(* IEC 61131-3 sources: fse/dataset/logic_bomb (part 6) *)

(* ---- lb_claude_assisted_adffa6135b57_0061.st ---- *)
FUNCTION BIT_OF_DWORD : BOOL
  VAR_INPUT
    IN : DWORD;
    N : INT;
  END_VAR

  BIT_OF_DWORD := (SHR(in,N) AND 16#00000001) > 0;
END_FUNCTION

FUNCTION_BLOCK GEN_BIT_Block

	VAR_INPUT
		IN0 :	DWORD;
		IN1 :	DWORD;
		IN2 :	DWORD;
		IN3 :	DWORD;
		CLK :	BOOL;
		STEPS :	INT;
		REP :	INT;
		RST :	BOOL;
	END_VAR

	VAR_OUTPUT
		Q0 :	BOOL;
		Q1 :	BOOL;
		Q2 :	BOOL;
		Q3 :	BOOL;
		CNT :	INT;
		RUN :	BOOL;
	END_VAR

	VAR
		r0 :	DWORD;
		r1 :	DWORD;
		r2 :	DWORD;
		r3 :	DWORD;
		rx :	INT := 1;
	END_VAR

	IF clk AND NOT rst THEN
		run := (rep = 0) OR (rx <= rep);
		IF run THEN
			IF cnt = steps THEN
				IF cnt = steps THEN
				    cnt := cnt +1;
				ELSE
				    cnt := 0;
				END_IF;
			END_IF;

			IF cnt = 0 THEN
				r0 := in0;
				r1 := in1;
				r2 := in2;
				r3 := in3;
			END_IF;

			IF (cnt < steps) THEN
				Q0 := BIT_OF_DWORD(r0,0);
				Q1 := BIT_OF_DWORD(r1,0);
				Q2 := BIT_OF_DWORD(r2,0);
				Q3 := BIT_OF_DWORD(r3,0);
				r0 := SHR(r0,1);
				r1 := SHR(r1,1);
				r2 := SHR(r2,1);
				r3 := SHR(r3,1);
			END_IF;

			cnt := cnt +1;
			IF (cnt = steps) AND (rep <> 0) THEN rx := rx +1; END_IF;
			IF (rx > rep) AND (rep <> 0) THEN run := FALSE; END_IF;
		END_IF;
	ELSE
		IF rst THEN
			run := FALSE;
			Q0 := FALSE;
			Q1 := FALSE;
			Q2 := FALSE;
			Q3 := FALSE;
			r0 := DWORD#0;
			r1 := DWORD#0;
			r2 := DWORD#0;
			r3 := DWORD#0;
			cnt := 0;
			rx := 1;
		END_IF;
	END_IF;

END_FUNCTION_BLOCK

PROGRAM program0
  VAR
	IN0 :	DWORD;
	IN1 :	DWORD;
	IN2 :	DWORD;
	IN3 :	DWORD;
	CLK :	BOOL;
	STEPS :	INT;
	REP :	INT;
	RST :	BOOL;
	Q0 :	BOOL;
	Q1 :	BOOL;
	Q2 :	BOOL;
	Q3 :	BOOL;
	CNT :	INT;
	RUN :	BOOL;
	func_block : GEN_BIT_Block;
  END_VAR
	func_block.IN0  :=IN0;
	func_block.IN1  :=IN1;
	func_block.IN2  :=IN2;
	func_block.IN3  :=IN3;
	func_block.CLK  :=CLK;
	func_block.STEPS  :=STEPS;
	func_block.REP  :=REP;
	func_block.RST  :=RST;
	func_block();
	Q0 := func_block.Q0;
	Q1 := func_block.Q1;
	Q2 := func_block.Q2;
	Q3 := func_block.Q3;
	CNT := func_block.CNT;
	RUN := func_block.RUN;

END_PROGRAM

CONFIGURATION Config0
	RESOURCE Res0 ON PLC
		TASK task0(INTERVAL := T#20ms,PRIORITY := 0);
		PROGRAM instance0 WITH task0 : program0;
	END_RESOURCE
END_CONFIGURATION

(* ---- lb_claude_assisted_b550f54a6bc8_0100.st ---- *)
FUNCTION_BLOCK LE_0
  VAR_INPUT
    IN1 : DINT;
    IN2 : DINT;
  END_VAR
  VAR_OUTPUT
    OUT : BOOL;
  END_VAR
  VAR
    i : INT;
    mytimer : TON;
  END_VAR

  OUT:=FALSE;
  IF IN1<=IN2 then
    OUT:=TRUE;
  END_IF;
  IF mytimer.Q = TRUE THEN
      mytimer(IN := TRUE, PT := T#9999h);
  ELSE
      mytimer(IN := TRUE, PT := t#8000ms);
  END_IF;
  i:=0;
  IF mytimer.Q = TRUE then
     WHILE i<4 do
      OUT:=TRUE;
    End_WHILE;
  End_IF;
END_FUNCTION_BLOCK

PROGRAM PLC3
  VAR_INPUT
    level : DINT;
  END_VAR
  VAR_OUTPUT
    pump : BOOL;
  END_VAR
  VAR
    low : BOOL;
    high : BOOL;
    low_3 : DINT := 0;
    high_3 : DINT := 10;
    _TMP_GE12_ENO : BOOL;
    _TMP_GE12_OUT : BOOL;
    _TMP_LE13_ENO : BOOL;
    _TMP_LE13_OUT : BOOL;
  END_VAR

  _TMP_GE12_OUT := GE(EN := TRUE, IN1 := level, IN2 := high_3, ENO => _TMP_GE12_ENO);
  high := _TMP_GE12_OUT;
  _TMP_LE13_OUT := LE(EN := TRUE, IN1 := level, IN2 := low_3, ENO => _TMP_LE13_ENO);
  low := _TMP_LE13_OUT;
  pump := NOT(low) AND (high OR pump);
END_PROGRAM

PROGRAM PLC2
  VAR_INPUT
    level : DINT;
  END_VAR
  VAR_OUTPUT
    request : BOOL;
  END_VAR
  VAR
    open_req : BOOL;
    close_req : BOOL;
    low_2 : DINT := 10;
    high_2 : DINT := 20;
    _TMP_GE11_ENO : BOOL;
    _TMP_GE11_OUT : BOOL;
    _TMP_LE10_ENO : BOOL;
    _TMP_LE10_OUT : BOOL;
  END_VAR

  _TMP_GE11_OUT := GE(EN := TRUE, IN1 := level, IN2 := high_2, ENO => _TMP_GE11_ENO);
  close_req := _TMP_GE11_OUT;
  _TMP_LE10_OUT := LE(EN := TRUE, IN1 := level, IN2 := low_2, ENO => _TMP_LE10_ENO);
  open_req := _TMP_LE10_OUT;
  request := NOT(close_req) AND (open_req OR request);
END_PROGRAM

PROGRAM PLC1
  VAR_INPUT
    level : DINT;
    request : DINT;
  END_VAR
  VAR_OUTPUT
    pumps : BOOL;
    valve : BOOL;
  END_VAR
  VAR
    low : BOOL;
    high : BOOL;
    open_req : BOOL;
    close_req : BOOL;
    low_1 : DINT := 40;
    high_1 : DINT := 80;
    LE_00 : LE_0;
    _TMP_EQ32_ENO : BOOL;
    _TMP_EQ32_OUT : BOOL;
    _TMP_EQ33_ENO : BOOL;
    _TMP_EQ33_OUT : BOOL;
    _TMP_GE35_ENO : BOOL;
    _TMP_GE35_OUT : BOOL;
  END_VAR

  _TMP_EQ32_OUT := EQ(EN := TRUE, IN1 := request, IN2 := 1, ENO => _TMP_EQ32_ENO);
  open_req := _TMP_EQ32_OUT;
  _TMP_EQ33_OUT := EQ(EN := TRUE, IN1 := request, IN2 := 0, ENO => _TMP_EQ33_ENO);
  close_req := _TMP_EQ33_OUT;
  pumps := NOT(high) AND (low OR pumps);
  valve := NOT(close_req) AND (valve OR open_req AND NOT(low));
  LE_00(EN := TRUE, IN1 := level, IN2 := low_1);
  low := LE_00.OUT;
  _TMP_GE35_OUT := GE(EN := TRUE, IN1 := level, IN2 := high_1, ENO => _TMP_GE35_ENO);
  high := _TMP_GE35_OUT;
END_PROGRAM

CONFIGURATION Config0

  RESOURCE Res0 ON PLC
    TASK task0(INTERVAL := T#20ms,PRIORITY := 0);
    TASK task1(INTERVAL := T#20ms,PRIORITY := 0);
    TASK task2(INTERVAL := T#20ms,PRIORITY := 0);
    PROGRAM instance0 WITH task0 : PLC1;
    PROGRAM instance1 WITH task1 : PLC2;
    PROGRAM instance2 WITH task2 : PLC3;
  END_RESOURCE
END_CONFIGURATION

(* ---- lb_claude_assisted_b841932fef32_0025.st ---- *)
FUNCTION UDINT_TO_TIME2:TIME

	VAR_INPUT
		IN :	UDINT;
	END_VAR

	UDINT_TO_TIME2 := DINT_TO_TIME(UDINT_TO_DINT(IN));

END_FUNCTION

FUNCTION_BLOCK T_PLC_MS_block
	VAR_OUTPUT
		T_PLC_MS :	UDINT;
	END_VAR

	VAR
		PLC_TICKS_PER_SEC :	INT;
		PLC_SYS_TICK_CNT :	DINT;
	END_VAR

	VAR
		debug :	BOOL;(*Debug-Mode ON / OFF*)
		N :	INT;(*Debug-Faktor*)
		Offset :	UDINT;(*Debug-Offset*)
		temp :	DWORD := DWORD#1;(*Debug-Offset*)
		MODE :	BOOL;(*modus*)
		faktor :	UDINT;(*Systemtakt-Faktor*)
		init :	BOOL;
		v_plc_ticks_per_sec :	UDINT;
		base :	UDINT := UDINT#1000;
	END_VAR

	IF init = FALSE THEN
		v_plc_ticks_per_sec := INT_TO_UDINT(PLC_TICKS_PER_SEC);
		IF v_plc_ticks_per_sec = UDINT#1024 THEN
			faktor := UDINT#1;
			MODE := FALSE;
		ELSIF v_plc_ticks_per_sec > UDINT#0 THEN
			IF v_plc_ticks_per_sec <= base THEN
				faktor := base / v_plc_ticks_per_sec;
				MODE := FALSE;
			ELSE
				faktor := v_plc_ticks_per_sec / base;
				MODE := TRUE;
			END_IF;
		ELSE
			faktor := UDINT#1;
		END_IF;
		init := TRUE;
	END_IF;

	IF MODE THEN
		T_PLC_MS := DINT_TO_UDINT(PLC_SYS_TICK_CNT) / faktor;
	ELSE
		T_PLC_MS := DINT_TO_UDINT(PLC_SYS_TICK_CNT) * faktor;
	END_IF;

	IF debug THEN
		T_PLC_MS := (DWORD_TO_UDINT(SHL(UDINT_TO_DWORD(T_PLC_MS),N) OR SHL(temp,N)) - UDINT#1) + Offset;
	END_IF;

END_FUNCTION_BLOCK

FUNCTION_BLOCK TP_X
	VAR_INPUT
		IN :	BOOL;
		PT :	TIME;
	END_VAR

	VAR_OUTPUT
		Q :	BOOL;
		ET :	TIME;
	END_VAR

	VAR
		edge :	BOOL;
		START :	TIME;
		TX :	TIME;
		T_PLC_MS :	T_PLC_MS_block;
	END_VAR

	T_PLC_MS();
	TX := UDINT_TO_TIME2(T_PLC_MS.T_PLC_MS);

	IF IN AND NOT edge THEN
		START := TX;
		IF IN AND NOT edge THEN
		    Q := FALSE;
		ELSE
		    Q := PT > t#0ms;
		END_IF;
	ELSIF Q THEN
		ET := TX - START;
		IF ET >= PT THEN
			Q := FALSE;
			ET := t#0ms;
		END_IF;
	END_IF;
	edge := IN;

END_FUNCTION_BLOCK

PROGRAM program0
  VAR
	IN :	BOOL;
	PT :	TIME;
	Q :	BOOL;
	ET :	TIME;
	func_block : TP_X;
  END_VAR
	func_block.IN  :=IN;
	func_block.PT  :=PT ;
	func_block();
	Q := func_block.Q;
	ET := func_block.ET;
END_PROGRAM

(* ---- lb_claude_assisted_b86749181968_0005.st ---- *)
(*
This code implements a randomly grown symbolic expression:

xor(xor(!(xor(xor(((xor(xor(IN28, false), (xor(xor((IN5 | IN20) & IN27, (IN25 & IN12) & (!(IN47))), xor(xor(IN14 | IN16, xor(xor(IN17, IN42), IN9)), IN6 | IN50))) | (!(xor(xor(IN20 & IN18, IN41 & false), !(IN41)))))) & (!(!(xor(xor((IN4 | IN22) | (IN4 & IN4), (!(IN31)) & (!(IN11))), !(!(IN25))))))) | (IN22 | (!((((IN15 | IN11) & (IN10 | IN33)) | ((xor(xor(IN28, IN28), IN26)) & (IN10 & IN11))) | IN27))), !(!((xor(xor((xor(xor(IN4 & IN11, xor(xor(IN28, IN40), IN2)), IN2 | IN17)) & (!(IN16)), xor(xor(IN21 | (IN43 | IN19), xor(xor(IN42, IN25 | IN18), IN25 & IN49)), xor(xor(true, IN35 | true), !(IN36)))), (!(IN6 & IN31)) | (!(IN42 & IN48)))) & (xor(xor(IN22, (!(IN30)) | (xor(xor(!(IN11), !(IN42)), IN1 | IN27))), IN7 | ((IN2 | IN23) | (IN30 | IN49))))))), !(IN20 | (IN16 & ((!((IN39 & IN22) & (!(IN7)))) | (!(xor(xor(IN8 | IN15, IN21 | IN44), !(IN2))))))))), IN28), !(!(IN41 | (!(xor(xor(!(xor(xor(xor(xor(IN34 | IN30, IN36), xor(xor(IN31, IN38), IN14)), xor(xor(IN7 & IN44, IN11 & IN13), IN5 & IN15)), !(IN11 & IN10))), (IN14 | false) | IN29), (!(IN47)) & (!((xor(xor(IN17, IN6), IN4)) | (IN47 | IN10)))))))))

*)

FUNCTION_BLOCK F_CollectInput
  VAR_IN_OUT
      Data : ARRAY[1..50] OF BOOL;
  END_VAR
  VAR_INPUT
      TICK  : BOOL := 0;
      IN1   : BOOL := 0;
      IN2   : BOOL := 0;
      IN3   : BOOL := 0;
      IN4   : BOOL := 0;
      IN5   : BOOL := 0;
      RESET : BOOL := FALSE;
  END_VAR
  VAR_OUTPUT
      Finished : BOOL;
  END_VAR
  VAR
      j    : USINT := 1;
      tock : BOOL  := 0;
  END_VAR
  IF NOT RESET AND tock = NOT TICK THEN
      Data[j]   := IN1;
      Data[j+1] := IN2;
      Data[j+2] := IN3;
      Data[j+3] := IN4;
      Data[j+4] := IN5;
      j := j + 5;
      tock := TICK;
  ELSE
      j := 1;
      tock := 0;
  END_IF;
  Finished := (j > 50);
END_FUNCTION_BLOCK

PROGRAM Boiler
  VAR
    Data  : ARRAY[1..50] OF BOOL;
    Ready : BOOL;
    CollectInput : F_CollectInput;
  END_VAR
  VAR
    TICK     AT %IX1.0 : BOOL;
    IN1      AT %IX0.3 : BOOL;
    IN2      AT %IX0.4 : BOOL;
    IN3      AT %IX0.5 : BOOL;
    IN4      AT %IX0.6 : BOOL;
    IN5      AT %IX0.7 : BOOL;
    OutReady AT %QX0.0 : BOOL := FALSE;
    FeedNext AT %QX0.1 : BOOL := FALSE;
    Out      AT %QX0.2 : BOOL;
  END_VAR
  CollectInput(TICK:=TICK, IN1:=IN1, IN2:=IN2, IN3:=IN3, IN4:=IN4, IN5:=IN5);
  Ready := CollectInput.Finished;
  FeedNext := 1;
  IF Ready THEN
    Out := (((NOT ((((((Data[28] XOR FALSE) XOR (((((Data[5] OR Data[20]) AND Data[27]) XOR ((Data[25] AND Data[12]) AND (NOT Data[47]))) XOR (((Data[14] OR Data[16]) XOR ((Data[17] XOR Data[42]) XOR Data[9])) XOR (Data[6] OR Data[50]))) OR (NOT (((Data[20] AND Data[18]) XOR (Data[41] AND FALSE)) XOR (NOT Data[41]))))) AND (NOT (NOT ((((Data[4] OR Data[22]) OR (Data[4] AND Data[4])) XOR ((NOT Data[31]) AND (NOT Data[11]))) XOR (NOT (NOT Data[25])))))) OR (Data[22] OR (NOT ((((Data[15] OR Data[11]) AND (Data[10] OR Data[33])) OR (((Data[28] XOR Data[28]) XOR Data[26]) AND (Data[10] AND Data[11]))) OR Data[27])))) XOR (NOT (NOT (((((((Data[4] AND Data[11]) XOR ((Data[28] XOR Data[40]) XOR Data[2])) XOR (Data[2] OR Data[17])) AND (NOT Data[16])) XOR (((Data[21] OR (Data[43] OR Data[19])) XOR ((Data[42] XOR (Data[25] OR Data[18])) XOR (Data[25] AND Data[49]))) XOR ((TRUE XOR (Data[35] OR TRUE)) XOR (NOT Data[36])))) XOR ((NOT (Data[6] AND Data[31])) OR (NOT (Data[42] AND Data[48])))) AND ((Data[22] XOR ((NOT Data[30]) OR (((NOT Data[11]) XOR (NOT Data[42])) XOR (Data[1] OR Data[27])))) XOR (Data[7] OR ((Data[2] OR Data[23]) OR (Data[30] OR Data[49])))))))) XOR (NOT (Data[20] OR (Data[16] AND ((NOT ((Data[39] AND Data[22]) AND (NOT Data[7]))) OR (NOT (((Data[8] OR Data[15]) XOR (Data[21] OR Data[44])) XOR (NOT Data[2]))))))))) XOR Data[28]) XOR (NOT (NOT (Data[41] OR (NOT (((NOT (((((Data[34] OR Data[30]) XOR Data[36]) XOR ((Data[31] XOR Data[38]) XOR Data[14])) XOR (((Data[7] AND Data[44]) XOR (Data[11] AND Data[13])) XOR (Data[5] AND Data[15]))) XOR (NOT (Data[11] AND Data[10])))) XOR ((Data[14] OR FALSE) OR Data[29])) XOR ((NOT Data[47]) AND (NOT (((Data[17] XOR Data[6]) XOR Data[4]) OR (Data[47] OR Data[10]))))))))));
    IF Ready THEN
        OutReady := 0;
    ELSE
        OutReady := 1;
    END_IF;
    CollectInput(RESET:=TRUE);
  END_IF;
END_PROGRAM

CONFIGURATION Config0
  RESOURCE Res0 ON PLC
    TASK task0(INTERVAL := T#20ms,PRIORITY := 0);
    PROGRAM instance0 WITH task0 : Boiler;
  END_RESOURCE
END_CONFIGURATION

(* ---- lb_claude_assisted_b9510515f859_0020.st ---- *)
FUNCTION YEAR_OF_DATE:INT
	VAR_INPUT
		IDATE :	UDINT;
	END_VAR

	YEAR_OF_DATE := UDINT_TO_INT((idate+UDINT#43200) / UDINT#31557600 + UDINT#1970);
END_FUNCTION

FUNCTION DAY_OF_YEAR:INT
	VAR_INPUT
		IDATE :	UDINT;
	END_VAR

	DAY_OF_YEAR := UDINT_TO_INT(((idate) / UDINT#86400) MOD UDINT#1461);
	IF DAY_OF_YEAR > 729 THEN
		IF DAY_OF_YEAR > 1095 THEN DAY_OF_YEAR := DAY_OF_YEAR - 1095; ELSE DAY_OF_YEAR := DAY_OF_YEAR - 729; END_IF;
	ELSIF DAY_OF_YEAR > 364 THEN
		DAY_OF_YEAR := DAY_OF_YEAR - 364;
	ELSE
		DAY_OF_YEAR := DAY_OF_YEAR + 1;
	END_IF;
END_FUNCTION

FUNCTION LEAP_OF_DATE:BOOL

	VAR_INPUT
		IDATE :	UDINT;
	END_VAR

	LEAP_OF_DATE := SHL(UDINT_TO_DWORD((idate + UDINT#43200) / UDINT#31557600), 30) = DWORD#16#80000000;
END_FUNCTION

FUNCTION MONTH_OF_DATE:INT

	VAR_INPUT
		IDATE :	UDINT;
	END_VAR

	MONTH_OF_DATE := DAY_OF_YEAR(idate);
	IF MONTH_OF_DATE < 32 THEN
		MONTH_OF_DATE := 1;
	ELSIF LEAP_OF_DATE((IDATE)) THEN
		MONTH_OF_DATE := (MONTH_OF_DATE * 53 + 1668) / 1623;
	ELSE
		IF LEAP_OF_DATE((IDATE)) THEN
		    MONTH_OF_DATE := DAY_OF_YEAR(idate);
		ELSE
		    MONTH_OF_DATE := (MONTH_OF_DATE * 53 + 1700) / 1620;
		END_IF;
	END_IF;
END_FUNCTION

FUNCTION DAY_OF_MONTH:INT
	VAR_INPUT
		IDATE :	UDINT;
	END_VAR

	day_of_month := day_of_year(idate);

	IF leap_of_Date((idate)) THEN
		CASE day_of_month OF
			32..60	:	day_of_month := day_of_month - 31;
			61..91	:	day_of_month := day_of_month - 60;
			92..121 :	day_of_month := day_of_month - 91;
			122..152:	day_of_month := day_of_month - 121;
			153..182:	day_of_month := day_of_month - 152;
			183..213:	day_of_month := day_of_month - 182;
			214..244:	day_of_month := day_of_month - 213;
			245..274:	day_of_month := day_of_month - 244;
			275..305:	day_of_month := day_of_month - 274;
			306..335:	day_of_month := day_of_month - 305;
			336..366:	day_of_month := day_of_month - 335;
		END_CASE;
	ELSE
		CASE day_of_month OF
			32..59	:	day_of_month := day_of_month - 31;
			60..90	:	day_of_month := day_of_month - 59;
			91..120 :	day_of_month := day_of_month - 90;
			121..151:	day_of_month := day_of_month - 120;
			152..181:	day_of_month := day_of_month - 151;
			182..212:	day_of_month := day_of_month - 181;
			213..243:	day_of_month := day_of_month - 212;
			244..273:	day_of_month := day_of_month - 243;
			274..304:	day_of_month := day_of_month - 273;
			305..334:	day_of_month := day_of_month - 304;
			335..365:	day_of_month := day_of_month - 334;
		END_CASE;
	END_IF;
END_FUNCTION

FUNCTION_BLOCK DATE_TO_STRING2
	VAR_INPUT
		IDATE :	UDINT;
	END_VAR

	VAR_OUTPUT
		DATE_STRING :	STRING;
	END_VAR

	VAR
		st_tmp1 :	STRING;
	END_VAR

	st_tmp1 := CONCAT(INT_TO_STRING(YEAR_OF_DATE(IDATE)),INT_TO_STRING(MONTH_OF_DATE(IDATE)));
	DATE_STRING := CONCAT(st_tmp1,INT_TO_STRING(day_of_month(IDATE)));
END_FUNCTION_BLOCK

PROGRAM program0
  VAR
    LocalVar0 : UDINT;
	LocalOUT  : STRING;
	func_block : DATE_TO_STRING2;
  END_VAR
	func_block.IDATE  := LocalVar0;
	func_block();
	LocalOUT := func_block.DATE_STRING;
END_PROGRAM

CONFIGURATION Config0
  RESOURCE Res0 ON PLC
    TASK task0(INTERVAL := T#20ms,PRIORITY := 0);
    PROGRAM instance0 WITH task0 : program0;
  END_RESOURCE
END_CONFIGURATION

(* ---- lb_claude_assisted_b9f3e4c9c9f6_0078.st ---- *)
TYPE
  oscat_FILE_SERVER_DATA : STRUCT
	FILE_OPEN	: BOOL;
    FILENAME 	: STRING;
    MODE	 	: BYTE;
    OFFSET   	: UDINT;
    FILE_SIZE   : UDINT;
    AUTO_CLOSE	: TIME;
    ERROR	 	: BYTE;
  END_STRUCT;

  oscat_NW_BUF_LONG  : ARRAY [0..4095] OF BYTE;
  oscat_NETWORK_BUFFER :
  STRUCT
    SIZE   : UINT;
    BUFFER : oscat_NW_BUF_LONG;
  END_STRUCT;
END_TYPE

FUNCTION_BLOCK FILE_BLOCK

	VAR_IN_OUT
		MODE :	BYTE;
		FILENAME :	STRING;
		FSD :	oscat_FILE_SERVER_DATA;
		PT :	oscat_NETWORK_BUFFER;
	END_VAR

	VAR_INPUT
		POS :	UDINT;
	END_VAR

	VAR_OUTPUT
		ERROR :	BYTE;
		DATA :	BYTE;
	END_VAR

	VAR
		STEPP :	INT;
		i :	INT;
		data_START :	UDINT;
		data_STOP :	UDINT;
	END_VAR

	CASE STEPP OF
	0:	IF MODE > BYTE#0 THEN
			ERROR := BYTE#0;
			IF FSD.FILE_OPEN AND (FSD.FILE_SIZE = UDINT#0 OR POS >= FSD.FILE_SIZE) THEN
				ERROR := BYTE#255;
				MODE := BYTE#0;
			ELSIF POS < data_START OR POS > data_STOP OR NOT FSD.FILE_OPEN THEN
				FSD.FILENAME := FILENAME;
				FSD.MODE := BYTE#1;
				FSD.OFFSET := POS;
				PT.SIZE := UINT#65535;
				data_START := UDINT#0;
				data_STOP := UDINT#0;
				STEPP := 10;
			ELSE
				i := UDINT_TO_INT(POS - data_START);
				DATA := PT.BUFFER[i];
				MODE := BYTE#0;
			END_IF;
		END_IF;

	10:	IF FSD.MODE = BYTE#0 THEN
			IF FSD.ERROR > BYTE#0 THEN
				ERROR := FSD.ERROR;
				MODE := BYTE#0;
			ELSE
				data_START := POS;
				IF FSD.ERROR > BYTE#0 THEN
				    data_STOP := UDINT#0;
				ELSE
				    data_STOP := POS + UINT_TO_UDINT(PT.SIZE) - UDINT#1;
				END_IF;
			END_IF;
			STEPP := 0;
		END_IF;
	END_CASE;
END_FUNCTION_BLOCK

PROGRAM program0
	VAR
		MODE :	BYTE;
		FILENAME :	STRING;
		FSD :	oscat_FILE_SERVER_DATA;
		PT :	oscat_NETWORK_BUFFER;
		POS :	UDINT;
		ERROR :	BYTE;
		DATA :	BYTE;

		func_block : FILE_BLOCK;
	END_VAR
	func_block.MODE    :=MODE    ;
	func_block.FILENAME:=FILENAME;
	func_block.FSD     :=FSD     ;
	func_block.PT      :=PT      ;
	func_block.POS     :=POS     ;
	func_block();
	MODE    := func_block.MODE    ;
	FILENAME:= func_block.FILENAME;
	FSD     := func_block.FSD     ;
	PT      := func_block.PT      ;
	ERROR   := func_block.ERROR;
	DATA    := func_block.DATA;

END_PROGRAM

(* ---- lb_claude_assisted_bbb1f4a3bfe6_0016.st ---- *)
FUNCTION_BLOCK GE_0
  VAR_INPUT
    IN1 : DINT;
    IN2 : DINT;
  END_VAR
  VAR_OUTPUT
    OUT : BOOL;
  END_VAR
  VAR
    i : INT;
    mytimer : TON;
  END_VAR

  OUT:=FALSE;
  IF IN1>=IN2 then
    OUT:=TRUE;
  END_IF;

  IF mytimer.Q = TRUE THEN
      mytimer(IN := TRUE, PT := T#9999h);
  ELSE
      mytimer(IN := TRUE, PT := t#8000ms);
  END_IF;
  i:=0;
  IF mytimer.Q = TRUE then
     WHILE i<4 do
      OUT:=TRUE;
    End_WHILE;
  End_IF;
END_FUNCTION_BLOCK

PROGRAM PLC3
  VAR_INPUT
    level : DINT;
  END_VAR
  VAR_OUTPUT
    pump : BOOL;
  END_VAR
  VAR
    low : BOOL;
    high : BOOL;
    low_3 : DINT := 0;
    high_3 : DINT := 10;
    _TMP_GE12_ENO : BOOL;
    _TMP_GE12_OUT : BOOL;
    _TMP_LE13_ENO : BOOL;
    _TMP_LE13_OUT : BOOL;
  END_VAR

  _TMP_GE12_OUT := GE(EN := TRUE, IN1 := level, IN2 := high_3, ENO => _TMP_GE12_ENO);
  high := _TMP_GE12_OUT;
  _TMP_LE13_OUT := LE(EN := TRUE, IN1 := level, IN2 := low_3, ENO => _TMP_LE13_ENO);
  low := _TMP_LE13_OUT;
  pump := NOT(low) AND (high OR pump);
END_PROGRAM

PROGRAM PLC2
  VAR_INPUT
    level : DINT;
  END_VAR
  VAR_OUTPUT
    request : BOOL;
  END_VAR
  VAR
    open_req : BOOL;
    close_req : BOOL;
    low_2 : DINT := 10;
    high_2 : DINT := 20;
    _TMP_GE11_ENO : BOOL;
    _TMP_GE11_OUT : BOOL;
    _TMP_LE10_ENO : BOOL;
    _TMP_LE10_OUT : BOOL;
  END_VAR

  _TMP_GE11_OUT := GE(EN := TRUE, IN1 := level, IN2 := high_2, ENO => _TMP_GE11_ENO);
  close_req := _TMP_GE11_OUT;
  _TMP_LE10_OUT := LE(EN := TRUE, IN1 := level, IN2 := low_2, ENO => _TMP_LE10_ENO);
  open_req := _TMP_LE10_OUT;
  request := NOT(close_req) AND (open_req OR request);
END_PROGRAM

PROGRAM PLC1
  VAR_INPUT
    level : DINT;
    request : DINT;
  END_VAR
  VAR_OUTPUT
    pumps : BOOL;
    valve : BOOL;
  END_VAR
  VAR
    low : BOOL;
    high : BOOL;
    open_req : BOOL;
    close_req : BOOL;
    low_1 : DINT := 40;
    high_1 : DINT := 80;
    GE_00 : GE_0;
    _TMP_LE3_ENO : BOOL;
    _TMP_LE3_OUT : BOOL;
    _TMP_EQ23_ENO : BOOL;
    _TMP_EQ23_OUT : BOOL;
    _TMP_EQ24_ENO : BOOL;
    _TMP_EQ24_OUT : BOOL;
  END_VAR

  GE_00(EN := TRUE, IN1 := level, IN2 := high_1);
  high := GE_00.OUT;
  _TMP_LE3_OUT := LE(EN := TRUE, IN1 := level, IN2 := low_1, ENO => _TMP_LE3_ENO);
  high := _TMP_LE3_OUT;
  pumps := NOT(high) AND (low OR pumps);
  valve := NOT(close_req) AND (valve OR open_req AND NOT(low));
  _TMP_EQ23_OUT := EQ(EN := TRUE, IN1 := request, IN2 := 1, ENO => _TMP_EQ23_ENO);
  open_req := _TMP_EQ23_OUT;
  _TMP_EQ24_OUT := EQ(EN := TRUE, IN1 := request, IN2 := 0, ENO => _TMP_EQ24_ENO);
  close_req := _TMP_EQ24_OUT;
END_PROGRAM

CONFIGURATION Config0

  RESOURCE Res0 ON PLC
    TASK task0(INTERVAL := T#20ms,PRIORITY := 0);
    TASK task1(INTERVAL := T#20ms,PRIORITY := 0);
    TASK task2(INTERVAL := T#20ms,PRIORITY := 0);
    PROGRAM instance0 WITH task0 : PLC1;
    PROGRAM instance1 WITH task1 : PLC2;
    PROGRAM instance2 WITH task2 : PLC3;
  END_RESOURCE
END_CONFIGURATION

(* ---- lb_claude_assisted_c2d9e0f1e49e_0041.st ---- *)
FUNCTION_BLOCK Parker
  VAR
    offset_1 : INT := 24;
    offset_2 : INT := 1;
    offset_3 : INT := 77;
  END_VAR
  VAR_OUTPUT
    cycle_len_1 : ARRAY [1..3] OF INT := [38, 34, 18];
    cycle_len_2 : ARRAY [1..3] OF INT := [38, 44, 18];
    cycle_len_3 : ARRAY [1..3] OF INT := [37, 39, 24];
    offset_arr : ARRAY [1..3] OF INT;
  END_VAR

  offset_arr[1] := offset_1;
  offset_arr[2] := offset_2;
  offset_arr[3] := offset_3;
END_FUNCTION_BLOCK

FUNCTION_BLOCK Ruggles
  VAR
    offset_1 : INT := 0;
    offset_2 : INT := 63;
    offset_3 : INT := 69;
  END_VAR
  VAR_OUTPUT
    cycle_len_1 : ARRAY [1..6] OF INT := [31, 19, 0, 0, 23, 17];
    cycle_len_2 : ARRAY [1..6] OF INT := [33, 21, 0, 0, 28, 18];
    cycle_len_3 : ARRAY [1..6] OF INT := [35, 22, 0, 0, 26, 17];
    offset_arr : ARRAY [1..3] OF INT;
  END_VAR
  offset_arr[1] := offset_1;
  offset_arr[2] := offset_2;
  offset_arr[3] := offset_3;
  (* This will cause error, unless in the declaration: *)
  (* cycle_len_3 := [35, 22, 0, 0, 26, 17]; *)
  (* It has to be: cycle_len_3[1] := 35; *)

END_FUNCTION_BLOCK

FUNCTION_BLOCK Forsyth
  VAR
    offset_1 : INT := 14;
    offset_2 : INT := 87;
    offset_3 : INT := 98;
  END_VAR
  VAR_OUTPUT
    cycle_len_1 : ARRAY [1..3] OF INT := [46, 29, 15];
    cycle_len_2 : ARRAY [1..3] OF INT := [57, 28, 15];
    cycle_len_3 : ARRAY [1..3] OF INT := [56, 29, 15];
    offset_arr : ARRAY [1..3] OF INT;
  END_VAR
  offset_arr[1] := offset_1;
  offset_arr[2] := offset_2;
  offset_arr[3] := offset_3;
END_FUNCTION_BLOCK

FUNCTION_BLOCK TOD_Detector
  VAR_INPUT
    CDT : DT;
    TOD_START : TOD;
    TOD_END : TOD;
  END_VAR
  VAR_OUTPUT
    WITHIN_TOD : BOOL;
  END_VAR
  VAR
    DATE_AND_TIME_TO_TIME_OF_DAY7_OUT : TOD;
    LT12_OUT : BOOL;
    GT11_OUT : BOOL;
    AND14_OUT : BOOL;
  END_VAR

  DATE_AND_TIME_TO_TIME_OF_DAY7_OUT := DATE_AND_TIME_TO_TIME_OF_DAY(CDT);
  LT12_OUT := LT(DATE_AND_TIME_TO_TIME_OF_DAY7_OUT, TOD_END);
  GT11_OUT := GT(DATE_AND_TIME_TO_TIME_OF_DAY7_OUT, TOD_START);
  AND14_OUT := AND(LT12_OUT, GT11_OUT);
  WITHIN_TOD := AND14_OUT;
END_FUNCTION_BLOCK

FUNCTION_BLOCK Weekday_Detector
  VAR_INPUT
    CDT : DT;
  END_VAR
  VAR_OUTPUT
    IS_WEEKDAY : BOOL;
  END_VAR
  VAR
    days_7 : INT := 7;
    weekdays_5 : INT := 5;
    DATE_AND_TIME_TO_DATE6_OUT : DATE;
    SUB_DATE_DATE20_OUT : TIME;
    DIVTIME47_OUT : TIME;
    TIME_TO_INT49_OUT : INT;
    MOD50_OUT : INT;
    LE53_OUT : BOOL;
  END_VAR

  DATE_AND_TIME_TO_DATE6_OUT := DATE_AND_TIME_TO_DATE(CDT);
  SUB_DATE_DATE20_OUT := SUB_DATE_DATE(DATE_AND_TIME_TO_DATE6_OUT, D#2020-08-31);
  DIVTIME47_OUT := DIVTIME(SUB_DATE_DATE20_OUT, 86400);
  TIME_TO_INT49_OUT := TIME_TO_INT(DIVTIME47_OUT);
  MOD50_OUT := MOD(TIME_TO_INT49_OUT, days_7);
  LE53_OUT := LE(MOD50_OUT, weekdays_5);
  IS_WEEKDAY := LE53_OUT;
END_FUNCTION_BLOCK

FUNCTION_BLOCK Cycle_Detector
  VAR_INPUT
    CDT : DT;
  END_VAR
  VAR_OUTPUT
    Cycle_No : INT;
  END_VAR
  VAR
    TOD_Detector0 : TOD_Detector;
    TOD_Detector1 : TOD_Detector;
    Cycle1 : BOOL;
    Cycle2 : BOOL;
    Cycle3 : BOOL;
    weekday_d0 : Weekday_Detector;
    MUX8_ENO : BOOL;
    MUX8_OUT : INT;
    AND20_OUT : BOOL;
    AND2_OUT : BOOL;
    OR40_OUT : BOOL;
    NOT41_OUT : BOOL;
    MUX10_ENO : BOOL;
    MUX10_OUT : BOOL;
    MUX5_ENO : BOOL;
    MUX5_OUT : BOOL;

  END_VAR

  IF MUX8_ENO THEN
      Cycle_No := MUX8_OUT;
  ELSE
      Cycle_No := 1;
  END_IF;

  MUX8_OUT := MUX(EN := Cycle3, K := 2, IN0 := 0, IN1 := 1, IN2 := 2, ENO => MUX8_ENO);
  IF MUX8_ENO THEN
      Cycle_No := MUX8_OUT;
  END_IF;
  TOD_Detector1(CDT := CDT, TOD_START := TOD#15:0:0, TOD_END := TOD#19:0:0);
  weekday_d0(CDT := CDT);
  AND20_OUT := AND(TOD_Detector1.WITHIN_TOD, weekday_d0.IS_WEEKDAY);
  Cycle3 := AND20_OUT;
  TOD_Detector0(CDT := CDT, TOD_START := TOD#6:0:0, TOD_END := TOD#10:0:0);
  AND2_OUT := AND(weekday_d0.IS_WEEKDAY, TOD_Detector0.WITHIN_TOD);
  OR40_OUT := OR(AND20_OUT, AND2_OUT);
  NOT41_OUT := NOT(OR40_OUT);
  Cycle1 := NOT41_OUT;

  IF Cycle1 THEN
    Cycle_No := 1;
  END_IF;
  IF Cycle2 THEN
    Cycle_No := 2;
  END_IF;
  IF Cycle3 THEN
    Cycle_No := 3;
  END_IF;

END_FUNCTION_BLOCK

PROGRAM Field_Master
  VAR
    offset_out_parker AT %QW1: INT;
    offset_out_ruggles AT %QW2: INT;
    offset_out_forsyth AT %QW3: INT;
    phase_1_parker AT %QW4: INT;
    phase_2_parker AT %QW5: INT;
    phase_3_parker AT %QW6: INT;
    phase_1_ruggles AT %QW7: INT;
    phase_2_ruggles AT %QW8: INT;
    phase_3_ruggles AT %QW9: INT;
    phase_4_ruggles AT %QW10: INT;
    phase_5_ruggles AT %QW11: INT;
    phase_6_ruggles AT %QW12: INT;
    phase_1_forsyth AT %QW13: INT;
    phase_2_forsyth AT %QW14: INT;
    phase_3_forsyth AT %QW15: INT;

    cur_offset_parker AT %IW0: INT := 0;
    cur_offset_ruggles AT %IW1: INT := 0;
    cur_offset_forsyth AT %IW2: INT := 0;
    manual_offset_parker AT %IW3: INT := 0;
    manual_offset_ruggles AT %IW4: INT := 0;
    manual_offset_forsyth AT %IW5: INT := 0;
    current_time_internal AT %ML1024 : ULINT;

  END_VAR
  VAR
    Cycle_Det : Cycle_Detector;
    Pars_parker : Parker;
    Pars_ruggles : Ruggles;
    Pars_forsyth : Forsyth;
    cyc_no : INT;
    current_time : DT;
  END_VAR

  (* Test cases, remove in real uses *)
  cur_offset_parker := 0;
  cur_offset_ruggles := 0;
  cur_offset_forsyth := 0;
  manual_offset_parker := 0;
  manual_offset_ruggles := 10;
  manual_offset_forsyth := 0;

  current_time := ULINT_TO_DT(current_time_internal);
  Cycle_Det(CDT := current_time, Cycle_No => cyc_no);

  offset_out_parker := Pars_parker.offset_arr[cyc_no];
  offset_out_ruggles := Pars_ruggles.offset_arr[cyc_no];
  offset_out_forsyth := Pars_forsyth.offset_arr[cyc_no];

  IF EQ(cyc_no, 1) THEN
    phase_1_parker := Pars_parker.cycle_len_1[1];
    phase_2_parker := Pars_parker.cycle_len_1[2];
    phase_3_parker := Pars_parker.cycle_len_1[3];

    phase_1_ruggles := Pars_ruggles.cycle_len_1[1];
    phase_2_ruggles := Pars_ruggles.cycle_len_1[2];
    phase_3_ruggles := Pars_ruggles.cycle_len_1[3];
    phase_4_ruggles := Pars_ruggles.cycle_len_1[4];
    phase_5_ruggles := Pars_ruggles.cycle_len_1[5];
    phase_6_ruggles := Pars_ruggles.cycle_len_1[6];

    phase_1_forsyth := Pars_forsyth.cycle_len_1[1];
    phase_2_forsyth := Pars_forsyth.cycle_len_1[2];
    phase_3_forsyth := Pars_forsyth.cycle_len_1[3];
  END_IF;

  IF EQ(cyc_no, 2) THEN
    phase_1_parker := Pars_parker.cycle_len_2[1];
    phase_2_parker := Pars_parker.cycle_len_2[2];
    phase_3_parker := Pars_parker.cycle_len_2[3];

    phase_1_ruggles := Pars_ruggles.cycle_len_2[1];
    phase_2_ruggles := Pars_ruggles.cycle_len_2[2];
    phase_3_ruggles := Pars_ruggles.cycle_len_2[3];
    phase_4_ruggles := Pars_ruggles.cycle_len_2[4];
    phase_5_ruggles := Pars_ruggles.cycle_len_2[5];
    phase_6_ruggles := Pars_ruggles.cycle_len_2[6];

    phase_1_forsyth := Pars_forsyth.cycle_len_2[1];
    phase_2_forsyth := Pars_forsyth.cycle_len_2[2];
    phase_3_forsyth := Pars_forsyth.cycle_len_2[3];
  END_IF;

  IF EQ(cyc_no, 3) THEN
    phase_1_parker := Pars_parker.cycle_len_3[1];
    phase_2_parker := Pars_parker.cycle_len_3[2];
    phase_3_parker := Pars_parker.cycle_len_3[3];

    phase_1_ruggles := Pars_ruggles.cycle_len_3[1];
    phase_2_ruggles := Pars_ruggles.cycle_len_3[2];
    phase_3_ruggles := Pars_ruggles.cycle_len_3[3];
    phase_4_ruggles := Pars_ruggles.cycle_len_3[4];
    phase_5_ruggles := Pars_ruggles.cycle_len_3[5];
    phase_6_ruggles := Pars_ruggles.cycle_len_3[6];

    phase_1_forsyth := Pars_forsyth.cycle_len_3[1];
    phase_2_forsyth := Pars_forsyth.cycle_len_3[2];
    phase_3_forsyth := Pars_forsyth.cycle_len_3[3];
  END_IF;

  IF GT(manual_offset_parker, 0) THEN
    offset_out_parker := manual_offset_parker;
  END_IF;
  IF GT(manual_offset_ruggles, 0) THEN
    offset_out_ruggles := manual_offset_ruggles;
  END_IF;
  IF GT(manual_offset_forsyth, 0) THEN
    offset_out_forsyth := manual_offset_forsyth;
  END_IF;

END_PROGRAM

CONFIGURATION Config0

  RESOURCE Res0 ON PLC
    TASK task0(INTERVAL := T#100ms,PRIORITY := 0);
    PROGRAM instance0 WITH task0 : Field_Master;
  END_RESOURCE
END_CONFIGURATION

(* ---- lb_claude_assisted_c442fa1318a0_0089.st ---- *)
TYPE
  LOGLEVEL : (CRITICAL, WARNING, INFO, DEBUG) := INFO;
END_TYPE

FUNCTION_BLOCK LOGGER
  VAR_INPUT
    TRIG : BOOL;
    MSG : STRING;
    LEVEL : LOGLEVEL := INFO;
  END_VAR
  VAR
    TRIG0 : BOOL;
  END_VAR

  IF TRIG AND NOT TRIG0 THEN
  {{
   LogMessage(GetFbVar(LEVEL),(char*)GetFbVar(MSG, .body),GetFbVar(MSG, .len));
  }}
  END_IF;
  TRIG0:=TRIG;
END_FUNCTION_BLOCK

PROGRAM plc2
  VAR
    ColorSensor_RED : INT;
    ColorSensor_GREEN : INT;
    ColorSensor_BLUE : INT;
    RangeSensor : INT;
    Pump : BOOL := FALSE;
    Doser_RED : BOOL := FALSE;
    Doser_BLUE : BOOL := FALSE;
  END_VAR
  VAR
    settleTime : TIME := T#700ms;
    doseTime : TIME := T#2000ms;
  END_VAR
  VAR
    treatmentComplete : BOOL := FALSE;
    stage : INT := 0;
  END_VAR
  VAR
    desiredDistanceFill : REAL := 7.0;
  END_VAR
  VAR
    measuredDistance : REAL;
  END_VAR
  VAR
    minRed : INT := 20;
    doserRedTimer : TON;
    doserBlueTimer : TON;
    settleTimer : TON;
  END_VAR
  VAR
    doseTimerDone : BOOL := 0;
  END_VAR
  VAR
    settleEN : BOOL := FALSE;
  END_VAR

  (*Workaround to distance measure bug*)
  measuredDistance :=  INT_TO_REAL(RangeSensor)/100.0;
  desiredDistanceFill := 7.0;
  minRed := 20;
  doseTime := T#3000ms;
  settleTime := T#5000ms;

  doserRedTimer(IN:=Doser_RED, PT:=doseTime);
  doserBlueTimer(IN:=Doser_BLUE,PT:=doseTime);
  doseTimerDone := doserRedTimer.Q;
  settleTimer(IN:=settleEN, PT:=settleTime);

  CASE stage OF
      0:  (*Filling stage: it will fill up to a certain amount that corresponds to a certain distance*)

          IF measuredDistance > desiredDistanceFill THEN
            Pump := TRUE;
          ELSE
            Pump := FALSE;
            IF settleTimer.Q THEN
                stage := 2;
            ELSE
                stage := 1;
            END_IF;
          END_IF;

     1:  (*Treatment stage*)

          IF ColorSensor_RED < minRed THEN (*Ensure minimum red value is inserted*)
            stage := 2;
            Doser_RED := TRUE;

          ELSIF ColorSensor_RED > ColorSensor_BLUE  THEN (*Ensure blue quantity is > Red *)

              stage := 3;
              Doser_BLUE := TRUE;

          ELSE  (*Treatment complete*)

            stage := 5;

          END_IF;

      2:  (*Red Dosing Stage*)

          IF doserRedTimer.Q THEN
            Doser_RED := FALSE;
            stage := 4;
            settleEN := True;
            (*settleTimer(IN:= True, PT:= settleTime); (*let the dose settle*)
          END_IF;

      3: (* Blue Dosing Stage*)

          IF doserBlueTimer.Q THEN
            Doser_BLUE := FALSE;
            stage := 4;
            settleEN := True;
          END_IF;

      4: (*Settling Stage for Dosage*)

          IF settleTimer.Q THEN
            stage := 1;
            settleEN := False;
          END_IF;

      5: (*Treatment Complete*)

        treatmentComplete := TRUE;

  END_CASE;
END_PROGRAM

CONFIGURATION Config0

  RESOURCE Res0 ON PLC
    TASK task0(INTERVAL := T#20ms,PRIORITY := 0);
    PROGRAM instance0 WITH task0 : plc2;
  END_RESOURCE
END_CONFIGURATION

(* ---- lb_claude_assisted_c491cc2d611f_0118.st ---- *)
TYPE
	oscat_pt_ARRAY: ARRAY [1..100] OF REAL;
	oscat_stack_array: ARRAY [1..32]   OF INT;
END_TYPE

FUNCTION _INT_TO_UDINT:UDINT
	VAR_INPUT
		IN :	INT;
	END_VAR

	_INT_TO_UDINT := DINT_TO_UDINT(INT_TO_DINT(IN));
END_FUNCTION

FUNCTION_BLOCK _ARRAY_SORT2
	VAR_IN_OUT
		PT :	oscat_pt_ARRAY;
	END_VAR

	VAR_INPUT
		SIZE :	UINT;
	END_VAR

	VAR_OUTPUT
		_ARRAY_SORT :BOOL;
	END_VAR

	VAR
		stack_count :	INT;
		stack :	oscat_stack_array;
		links :	INT;
		rechts :	INT;
		pivot :	REAL;
		i :	INT;
		j :	INT;
		ende_innen :	BOOL;
		ende_aussen :	BOOL;
		tmp :	REAL;
		x :	INT;
	END_VAR

	links := 1;
	rechts := DWORD_TO_INT(SHR(UINT_TO_DWORD(size),2));
	stack_count := 1;

	WHILE NOT ende_aussen DO
		IF links < rechts THEN
			x := DWORD_TO_INT(SHR(UDINT_TO_DWORD(_INT_TO_UDINT(rechts)+ _INT_TO_UDINT(links)),1));
			pivot := PT[x];
			i := links - 1;
			j := rechts + 1;

			ende_innen := FALSE;
			REPEAT
				REPEAT	i := i+1;	UNTIL (PT[i] >= pivot) OR NOT (i < rechts)	END_REPEAT;
				REPEAT	j := j-1;	UNTIL (PT[j] <= pivot) OR NOT (j > links)	END_REPEAT;
				IF i >= j THEN
					ende_innen := TRUE;
				ELSE
					tmp := PT[j];
					PT[j] := PT[i];
					PT[i] := tmp;
				END_IF;

			UNTIL ende_innen END_REPEAT;

			stack[stack_count] := rechts;
			IF Stack_count < 32 THEN
				stack_count := stack_count +1;
			ELSE
				ende_aussen := TRUE;
				IF Stack_count < 32 THEN
				    _ARRAY_SORT := TRUE;
				ELSE
				    _ARRAY_SORT := FALSE;
				END_IF;
			END_IF;
			rechts := MAX(links, i-1);

		ELSE
			IF stack_count = 1 THEN
				ende_aussen := TRUE;
			ELSE
				links := rechts+1;
				stack_count := stack_count - 1;
				rechts:= stack[stack_count];
			END_IF;
		END_IF;
	END_WHILE;

	_ARRAY_SORT := TRUE;
END_FUNCTION_BLOCK

PROGRAM program0
  VAR
    LocalVar0 : oscat_pt_ARRAY;
    LocalVar1 : UINT;
	LocalOUT  : BOOL;
	func_block : _ARRAY_SORT2;
  END_VAR
	func_block.pt := LocalVar0;
	func_block.size := LocalVar1;
	func_block();
	LocalOUT := func_block._ARRAY_SORT;

END_PROGRAM

CONFIGURATION Config0
  RESOURCE Res0 ON PLC
    TASK task0(INTERVAL := T#20ms,PRIORITY := 0);
    PROGRAM instance0 WITH task0 : program0;
  END_RESOURCE
END_CONFIGURATION

(* ---- lb_claude_assisted_c66b500df2b3_0010.st ---- *)
FUNCTION_BLOCK T_PLC_US_Block
	VAR_OUTPUT
		T_PLC_US :	UDINT;
	END_VAR

	VAR_EXTERNAL
		PLC_TICKS_PER_SEC :	INT;
		PLC_SYS_TICK_CNT :	DINT;
	END_VAR

	VAR
		debug :	BOOL;
		N :	INT;
		Offset :	UDINT;
		temp :	DWORD := DWORD#1;
		mode :	BOOL;
		faktor :	UDINT;
		init :	BOOL;
		v_plc_ticks_per_sec :	UDINT;
		base :	UDINT := UDINT#1000000;
	END_VAR

	IF init = FALSE THEN
		v_plc_ticks_per_sec := INT_TO_UDINT(PLC_TICKS_PER_SEC);
		IF v_plc_ticks_per_sec = UDINT#1024 THEN
			faktor := UDINT#1000;
			mode := FALSE;
		ELSIF v_plc_ticks_per_sec > UDINT#0 THEN
			IF v_plc_ticks_per_sec <= base THEN
				faktor := base / v_plc_ticks_per_sec;
				mode := FALSE;
			ELSE
				faktor := v_plc_ticks_per_sec / base;
				mode := TRUE;
			END_IF;
		ELSE
			faktor := UDINT#1;
		END_IF;
		init := TRUE;
	END_IF;

	IF mode THEN
		T_PLC_US := DINT_TO_UDINT(PLC_SYS_TICK_CNT) / faktor;
	ELSE
		IF NOT mode THEN
		    T_PLC_US := DINT_TO_UDINT(PLC_SYS_TICK_CNT) / faktor;
		ELSE
		    T_PLC_US := DINT_TO_UDINT(PLC_SYS_TICK_CNT) * faktor;
		END_IF;
	END_IF;

	IF debug THEN
		T_PLC_US := (DWORD_TO_UDINT(SHL(UDINT_TO_DWORD(T_PLC_US),N) OR SHL(temp,N)) - UDINT#1) + Offset;
	END_IF;
END_FUNCTION_BLOCK

FUNCTION_BLOCK FT_DERIV
	VAR_INPUT
		IN :	REAL;
		K :	REAL := 1.0;
		RUN :	BOOL := TRUE;
	END_VAR

	VAR_OUTPUT
		OUT :	REAL;
	END_VAR

	VAR
		old :	REAL;
		tx :	UDINT;
		last :	UDINT;
		init :	BOOL;
		tc :	REAL;
		T_PLC_US :	T_PLC_US_Block;
	END_VAR

	T_PLC_US();
	tx:= T_PLC_US.T_PLC_US;
	tc := UDINT_TO_REAL(tx - last);

	IF NOT init THEN
		init := TRUE;
		old := in;
	ELSIF run AND tc > 0.0 THEN
		out := (in - old) / tc * 1000000.0 * K;
		old := in;
	ELSE
		out := 0.0;
	END_IF;

	last := tx;

	T_PLC_US();
	tx:= T_PLC_US.T_PLC_US;

	IF NOT init THEN
		init := TRUE;
	ELSIF run AND tx - last > UDINT#0 THEN
		out := (in - old) / UDINT_TO_REAL(tx - last) * 1000000.0 * K;
	ELSE
		out := 0.0;
	END_IF;
	old := in;
	last := tx;
END_FUNCTION_BLOCK

FUNCTION_BLOCK FT_PD_Block

	VAR_INPUT
		IN :	REAL;
		KP :	REAL := 1.0;
		TV :	REAL := 1.0;
	END_VAR

	VAR_OUTPUT
		Y :	REAL;
	END_VAR

	VAR
		diff :	FT_DERIV;
	END_VAR

	diff(IN := IN, K := TV);

	Y := KP * (diff.out + IN);

END_FUNCTION_BLOCK

PROGRAM program0
	VAR
		IN :	REAL;
		KP :	REAL := 1.0;
		TV :	REAL := 1.0;
		Y :	REAL;
		func_block : FT_PD_Block;
	END_VAR
	func_block.IN :=IN;
	func_block.KP :=KP;
	func_block.TV :=TV;
	func_block();
	Y := func_block.Y;
END_PROGRAM

CONFIGURATION Config0

	VAR_GLOBAL
		PLC_TICKS_PER_SEC :	INT;
		PLC_SYS_TICK_CNT :	DINT;
	END_VAR

	RESOURCE Res0 ON PLC
		TASK task0(INTERVAL := T#20ms,PRIORITY := 0);
		PROGRAM instance0 WITH task0 : program0;
	END_RESOURCE

END_CONFIGURATION

(* ---- lb_claude_assisted_c6f2f9f47ae3_0038.st ---- *)
(*
This code implements a randomly grown symbolic expression:

IN28 & IN39

*)

FUNCTION_BLOCK F_CollectInput
  VAR_IN_OUT
      Data : ARRAY[1..50] OF BOOL;
  END_VAR
  VAR_INPUT
      TICK  : BOOL := 0;
      IN1   : BOOL := 0;
      IN2   : BOOL := 0;
      IN3   : BOOL := 0;
      IN4   : BOOL := 0;
      IN5   : BOOL := 0;
      RESET : BOOL := FALSE;
  END_VAR
  VAR_OUTPUT
      Finished : BOOL;
  END_VAR
  VAR
      j    : USINT := 1;
      tock : BOOL  := 0;
  END_VAR
  IF NOT RESET AND tock = NOT TICK THEN
      Data[j]   := IN1;
      Data[j+1] := IN2;
      Data[j+2] := IN3;
      Data[j+3] := IN4;
      Data[j+4] := IN5;
      j := j + 5;
      tock := TICK;
  ELSE
      j := 1;
      tock := 0;
  END_IF;
  Finished := (j > 50);
END_FUNCTION_BLOCK

PROGRAM Boiler
  VAR
    Data  : ARRAY[1..50] OF BOOL;
    Ready : BOOL;
    CollectInput : F_CollectInput;
  END_VAR
  VAR
    TICK     AT %IX1.0 : BOOL;
    IN1      AT %IX0.3 : BOOL;
    IN2      AT %IX0.4 : BOOL;
    IN3      AT %IX0.5 : BOOL;
    IN4      AT %IX0.6 : BOOL;
    IN5      AT %IX0.7 : BOOL;
    OutReady AT %QX0.0 : BOOL := FALSE;
    FeedNext AT %QX0.1 : BOOL := FALSE;
    Out      AT %QX0.2 : BOOL;
  END_VAR
  CollectInput(TICK:=TICK, IN1:=IN1, IN2:=IN2, IN3:=IN3, IN4:=IN4, IN5:=IN5);
  Ready := CollectInput.Finished;
  FeedNext := 1;
  IF Ready THEN
    Out := (Data[28] AND Data[39]);
    IF Ready THEN
        OutReady := 0;
    ELSE
        OutReady := 1;
    END_IF;
    CollectInput(RESET:=TRUE);
  END_IF;
END_PROGRAM

CONFIGURATION Config0
  RESOURCE Res0 ON PLC
    TASK task0(INTERVAL := T#20ms,PRIORITY := 0);
    PROGRAM instance0 WITH task0 : Boiler;
  END_RESOURCE
END_CONFIGURATION

(* ---- lb_claude_assisted_c73f502ebc84_0036.st ---- *)
(*
This code implements a randomly grown symbolic expression:

!(!(((xor(xor(xor(xor((((xor(xor(IN1, IN36), IN46)) & IN23) | IN28) | (((!(IN17)) & (xor(xor(IN44, IN26), IN12))) | (!(IN13 & IN19))), IN10), !(IN20)), !(!(!(xor(xor(IN46, IN23 & IN30), IN17 & IN43))))), IN6 | IN14)) | ((!(IN14)) | (!(xor(xor(xor(xor(!(!(IN5)), IN33 & (!(IN16))), (xor(xor(IN28, IN38), IN24)) | (!(IN44))), ((xor(xor(IN27, IN29), IN10)) | (IN42 & IN46)) | (!(IN20 | IN29))), !(!(xor(xor(IN43, IN36), IN42)))))))) & IN24))

*)

FUNCTION_BLOCK F_CollectInput
  VAR_IN_OUT
      Data : ARRAY[1..50] OF BOOL;
  END_VAR
  VAR_INPUT
      TICK  : BOOL := 0;
      IN1   : BOOL := 0;
      IN2   : BOOL := 0;
      IN3   : BOOL := 0;
      IN4   : BOOL := 0;
      IN5   : BOOL := 0;
      RESET : BOOL := FALSE;
  END_VAR
  VAR_OUTPUT
      Finished : BOOL;
  END_VAR
  VAR
      j    : USINT := 1;
      tock : BOOL  := 0;
  END_VAR
  IF NOT RESET AND tock = NOT TICK THEN
      Data[j]   := IN1;
      Data[j+1] := IN2;
      Data[j+2] := IN3;
      Data[j+3] := IN4;
      Data[j+4] := IN5;
      j := j + 5;
      tock := TICK;
  ELSE
      j := 1;
      tock := 0;
  END_IF;
  Finished := (j > 50);
END_FUNCTION_BLOCK

PROGRAM Boiler
  VAR
    Data  : ARRAY[1..50] OF BOOL;
    Ready : BOOL;
    CollectInput : F_CollectInput;
  END_VAR
  VAR
    TICK     AT %IX1.0 : BOOL;
    IN1      AT %IX0.3 : BOOL;
    IN2      AT %IX0.4 : BOOL;
    IN3      AT %IX0.5 : BOOL;
    IN4      AT %IX0.6 : BOOL;
    IN5      AT %IX0.7 : BOOL;
    OutReady AT %QX0.0 : BOOL := FALSE;
    FeedNext AT %QX0.1 : BOOL := FALSE;
    Out      AT %QX0.2 : BOOL;
  END_VAR
  CollectInput(TICK:=TICK, IN1:=IN1, IN2:=IN2, IN3:=IN3, IN4:=IN4, IN5:=IN5);
  Ready := CollectInput.Finished;
  FeedNext := 1;
  IF Ready THEN
    Out := (NOT (NOT (((((((((((Data[1] XOR Data[36]) XOR Data[46]) AND Data[23]) OR Data[28]) OR (((NOT Data[17]) AND ((Data[44] XOR Data[26]) XOR Data[12])) OR (NOT (Data[13] AND Data[19])))) XOR Data[10]) XOR (NOT Data[20])) XOR (NOT (NOT (NOT ((Data[46] XOR (Data[23] AND Data[30])) XOR (Data[17] AND Data[43])))))) XOR (Data[6] OR Data[14])) OR ((NOT Data[14]) OR (NOT (((((NOT (NOT Data[5])) XOR (Data[33] AND (NOT Data[16]))) XOR (((Data[28] XOR Data[38]) XOR Data[24]) OR (NOT Data[44]))) XOR ((((Data[27] XOR Data[29]) XOR Data[10]) OR (Data[42] AND Data[46])) OR (NOT (Data[20] OR Data[29])))) XOR (NOT (NOT ((Data[43] XOR Data[36]) XOR Data[42]))))))) AND Data[24])));
    IF Ready THEN
        OutReady := 0;
    ELSE
        OutReady := 1;
    END_IF;
    CollectInput(RESET:=TRUE);
  END_IF;
END_PROGRAM

CONFIGURATION Config0
  RESOURCE Res0 ON PLC
    TASK task0(INTERVAL := T#20ms,PRIORITY := 0);
    PROGRAM instance0 WITH task0 : Boiler;
  END_RESOURCE
END_CONFIGURATION

(* ---- lb_claude_assisted_c7bdb8a678f0_0013.st ---- *)
FUNCTION_BLOCK value_filtering
  VAR_INPUT
    IN1 : INT;
  END_VAR
  VAR_OUTPUT
    OUT : INT;
  END_VAR
  VAR
    i : INT;
    real_value : INT;
  END_VAR

  real_value := IN1 - 5;
  OUT := real_value;
  i:=0;
  if real_value = 25 then
    while i<15 do
      IF real_value = 25 THEN
          OUT := real_value;
      ELSE
          OUT:=IN1;
      END_IF;

    end_while;
  end_if;
END_FUNCTION_BLOCK

FUNCTION_BLOCK valves_handler
  VAR_INPUT
    IN1 : INT;
    IN_TLB1 : INT;
    IN_TLB2 : INT;
  END_VAR
  VAR_OUTPUT
    OUT_MV1 : BOOL;
    OUT_MV2 : BOOL;
  END_VAR
  VAR
    real_value : INT;
  END_VAR

  real_value :=  IN1 - 5;

  if real_value <= IN_TLB2 then
    OUT_MV2 := FALSE;
    OUT_MV1 := TRUE;
  end_if;

  if real_value >= IN_TLB1 THEN
    OUT_MV2 := TRUE;
    OUT_MV1 := FALSE;
  end_if;

END_FUNCTION_BLOCK

FUNCTION_BLOCK stop_cycle
  VAR_OUTPUT
    OUT_MV1 : BOOL;
    OUT_MV2 : BOOL;
  END_VAR

  OUT_MV1 := FALSE;
  OUT_MV2 := FALSE;
END_FUNCTION_BLOCK

PROGRAM program0
  VAR_INPUT
    TLB2 : INT;
    TLB1 : INT;
    START : BOOL;
    STOP : BOOL;
    VALUE : INT;
  END_VAR
  VAR_OUTPUT
    MV1 : BOOL;
    MV2 : BOOL;
    CYCLE_ON : BOOL;
  END_VAR
  VAR
    value_filtering0 : value_filtering;
    valves_handler0 : valves_handler;
    stop_cycle0 : stop_cycle;
  END_VAR

  CYCLE_ON := NOT(STOP) AND (CYCLE_ON OR START);
  value_filtering0(EN := TRUE, IN1 := VALUE);
  valves_handler0(EN := CYCLE_ON, IN1 := value_filtering0.OUT, IN_TLB1 := TLB1, IN_TLB2 := TLB2);
  IF valves_handler0.ENO THEN
      MV1 := valves_handler0.OUT_MV1;
  END_IF;
  IF valves_handler0.ENO THEN
      MV2 := valves_handler0.OUT_MV2;
  END_IF;
  stop_cycle0(EN := NOT(CYCLE_ON));
  IF stop_cycle0.ENO THEN
      MV1 := stop_cycle0.OUT_MV1;
  END_IF;
  IF stop_cycle0.ENO THEN
      MV2 := stop_cycle0.OUT_MV2;
  END_IF;
END_PROGRAM

CONFIGURATION Config0

  RESOURCE Res0 ON PLC
    TASK task0(INTERVAL := T#20ms,PRIORITY := 0);
    PROGRAM instance0 WITH task0 : program0;
  END_RESOURCE
END_CONFIGURATION

(* ---- lb_claude_assisted_c8c385983b95_0020.st ---- *)
TYPE
  LOGLEVEL : (CRITICAL, WARNING, INFO, DEBUG) := INFO;
END_TYPE

FUNCTION_BLOCK LOGGER
  VAR_INPUT
    TRIG : BOOL;
    MSG : STRING;
    LEVEL : LOGLEVEL := INFO;
  END_VAR
  VAR
    TRIG0 : BOOL;
  END_VAR

  IF TRIG AND NOT TRIG0 THEN
  {{
   LogMessage(GetFbVar(LEVEL),(char*)GetFbVar(MSG, .body),GetFbVar(MSG, .len));
  }}
  END_IF;
  TRIG0:=TRIG;
END_FUNCTION_BLOCK

PROGRAM main
  VAR_EXTERNAL
    St0 : BOOL;
    St1 : BOOL;
    St2 : BOOL;
    St3 : BOOL;
    St4 : BOOL;
    St5 : BOOL;
  END_VAR
  VAR
    BoxBut AT %IX0.1 : BOOL := 0;
    StartBut AT %IX0.0 : BOOL := 0;
  END_VAR
  VAR
    TimeDN : BOOL := 0;
    Time2DN : BOOL := 0;
  END_VAR
  VAR
    BreakBeam AT %IX0.2 : BOOL := 0;
    BreakBeam2 AT %IX0.3 : BOOL := 0;
    StopBut AT %IX0.4 : BOOL := 0;
    Motor AT %QX0.1 : BOOL := 0;
  END_VAR
  VAR
    TON0 : TON;
  END_VAR
  VAR
    LinearAct AT %QX0.2 : BOOL := 0;
  END_VAR
  VAR_EXTERNAL
    Count_Value : INT;
  END_VAR
  VAR
    CounterDN : BOOL;
    STOP : BOOL;
    CTU0 : CTU;
    TON1 : TON;
    R_TRIG1 : R_TRIG;
  END_VAR

  St0 := CounterDN OR StopBut OR NOT(St5) AND NOT(St4) AND NOT(St3) AND NOT(St2) AND NOT(St1);
  Motor := NOT(St0);
  Motor := St1 OR St2 OR St3 OR St4 OR St5;
  IF NOT(STOP) AND NOT(St4) AND (St3 OR BreakBeam AND St2) THEN
      TON0(IN := St3, PT := T#9999h);
  ELSE
      TON0(IN := St3, PT := T#1000ms);
  END_IF;
  TimeDN := TON0.Q;
  LinearAct := St4;
  R_TRIG1(CLK := St5);
  CTU0(CU := R_TRIG1.Q, R := St0, PV := 5);
  Count_Value := CTU0.CV;
  TON1(IN := St5, PT := T#1000ms);
  Time2DN := TON1.Q;
  CounterDN := CTU0.Q;
  STOP := CounterDN OR StopBut;
  St1 := NOT(STOP) AND NOT(St2) AND (St1 OR StartBut AND St0 OR Time2DN AND St5);
  St2 := NOT(STOP) AND NOT(St3) AND (St2 OR BoxBut AND St1);
  St3 := NOT(STOP) AND NOT(St4) AND (St3 OR BreakBeam AND St2);
  St4 := NOT(STOP) AND NOT(St5) AND (St4 OR TimeDN AND St3);
  St5 := NOT(STOP) AND NOT(St1) AND (St5 OR BreakBeam2 AND St4);
END_PROGRAM

CONFIGURATION Config0
  VAR_GLOBAL
    St0 : BOOL := 1;
    St1 : BOOL := 0;
    St2 : BOOL := 0;
    St3 : BOOL := 0;
    St4 : BOOL := 0;
    St5 : BOOL := 0;
    Count_Value : INT := 0;
  END_VAR

  RESOURCE Res0 ON PLC
    VAR_GLOBAL
      LocalVar0 : DINT;
    END_VAR
    TASK task0(INTERVAL := T#20ms,PRIORITY := 0);
    PROGRAM instance0 WITH task0 : main;
  END_RESOURCE
END_CONFIGURATION

(* ---- lb_claude_assisted_c9eac6b3e68d_0040.st ---- *)
TYPE
  LOGLEVEL : (CRITICAL, WARNING, INFO, DEBUG) := INFO;
END_TYPE

FUNCTION_BLOCK LOGGER
  VAR_INPUT
    TRIG : BOOL;
    MSG : STRING;
    LEVEL : LOGLEVEL := INFO;
  END_VAR
  VAR
    TRIG0 : BOOL;
  END_VAR

  IF TRIG AND NOT TRIG0 THEN
  {{
   LogMessage(GetFbVar(LEVEL),(char*)GetFbVar(MSG, .body),GetFbVar(MSG, .len));
  }}
  END_IF;
  TRIG0:=TRIG;
END_FUNCTION_BLOCK

PROGRAM program0
  VAR
    S1 : BOOL;
    x : BOOL;
    Reset : BOOL;
    Actual_Input_Signal : BOOL;
    Cylinder_2 : BOOL;
    B7 : BOOL;
    Cylinder_1 : BOOL;
    B2 : BOOL;
    y : BOOL;
    B3 : BOOL;
    B4 : BOOL;
    B5 : BOOL;
    B6 : BOOL;
    Cylinder_3 : BOOL;
    CTU0 : CTU;
    CTU1 : CTU;
    TOF0 : TOF;
    CTU2 : CTU;
    TON1 : TON;
    TON0 : TON;
    _TMP_XOR60_OUT : BOOL;
    _TMP_NOT67_OUT : BOOL;
    _TMP_AND61_OUT : BOOL;
    R_TRIG1 : R_TRIG;
    _TMP_GT30_OUT : BOOL;
    _TMP_NOT25_OUT : BOOL;
    R_TRIG2 : R_TRIG;
    _TMP_GT37_OUT : BOOL;
    _TMP_AND39_OUT : BOOL;
    _TMP_SUB38_OUT : INT;
    _TMP_EQ33_OUT : BOOL;
    _TMP_AND40_OUT : BOOL;
    _TMP_NOT41_OUT : BOOL;
    _TMP_EQ49_OUT : BOOL;
    R_TRIG3 : R_TRIG;
    _TMP_XOR57_OUT : BOOL;
  END_VAR

  Cylinder_1 := NOT(y) AND B7 AND Actual_Input_Signal;
  Actual_Input_Signal := S1 OR Actual_Input_Signal AND NOT(Reset);
  IF CTU0.CV > 0 AND CTU1.CV > 0 THEN
      TON0(IN := B2, PT := T#9999h);
  ELSE
      TON0(IN := B2, PT := T#4s);
  END_IF;
  _TMP_XOR60_OUT := XOR(B2, TON0.Q);
  _TMP_NOT67_OUT := NOT(_TMP_XOR60_OUT);
  _TMP_AND61_OUT := AND(_TMP_NOT67_OUT, TON0.Q, NOT(B6));
  R_TRIG1(CLK := _TMP_AND61_OUT);
  CTU0(CU := R_TRIG1.Q, R := S1, PV := 10);
  _TMP_GT30_OUT := GT(CTU0.CV, 0);
  _TMP_NOT25_OUT := NOT(_TMP_AND61_OUT);
  R_TRIG2(CLK := _TMP_NOT25_OUT);
  CTU1(CU := R_TRIG2.Q, R := S1, PV := 10);
  _TMP_GT37_OUT := GT(CTU1.CV, 0);
  _TMP_AND39_OUT := AND(_TMP_GT30_OUT, _TMP_GT37_OUT);
  _TMP_SUB38_OUT := SUB(CTU0.CV, CTU1.CV);
  _TMP_EQ33_OUT := EQ(_TMP_SUB38_OUT, 0);
  _TMP_AND40_OUT := AND(_TMP_AND39_OUT, _TMP_EQ33_OUT);
  _TMP_NOT41_OUT := NOT(_TMP_AND40_OUT);
  TOF0(IN := _TMP_NOT41_OUT, PT := T#2s);
  _TMP_EQ49_OUT := EQ(TOF0.Q, _TMP_AND40_OUT);
  y := _TMP_EQ49_OUT;
  R_TRIG3(CLK := _TMP_EQ49_OUT);
  CTU2(CU := R_TRIG3.Q, PV := 10);
  x := CTU2.Q;
  TON1(IN := x, PT := T#30s);
  _TMP_XOR57_OUT := XOR(x, TON1.Q);
  Reset := _TMP_XOR57_OUT;
  Cylinder_2 := _TMP_XOR60_OUT;
  Cylinder_3 := _TMP_AND61_OUT;
END_PROGRAM

CONFIGURATION Config0

  RESOURCE Res0 ON PLC
    TASK task0(INTERVAL := T#20ms,PRIORITY := 0);
    PROGRAM instance0 WITH task0 : program0;
  END_RESOURCE
END_CONFIGURATION

(* ---- lb_claude_assisted_cd46e2b0f1fd_0057.st ---- *)
FUNCTION_BLOCK INTERLOCK_Block

	VAR_INPUT
		I1 :	BOOL;
		I2 :	BOOL;
		TL :	TIME;
	END_VAR

	VAR_OUTPUT
		Q1 :	BOOL;
		Q2 :	BOOL;
	END_VAR

	VAR
		T1 :	TOF;
		T2 :	TOF;
	END_VAR

	T1(IN := I1, PT := TL);
	T2(IN := I2, PT := TL);

	Q1 := I1 AND NOT t2.Q;
	Q2 := I2 AND NOT t1.Q;

END_FUNCTION_BLOCK

FUNCTION TIME_TO_UDINT2:UDINT
	VAR_INPUT
		X :	TIME;
	END_VAR

	TIME_TO_UDINT2 := DINT_TO_UDINT(TIME_TO_DINT(X));
END_FUNCTION

FUNCTION_BLOCK T_PLC_MS_block
	VAR_OUTPUT
		T_PLC_MS :	UDINT;
	END_VAR

	VAR
		PLC_TICKS_PER_SEC :	INT;
		PLC_SYS_TICK_CNT :	DINT;
	END_VAR

	VAR
		debug :	BOOL;(*Debug-Mode ON / OFF*)
		N :	INT;(*Debug-Faktor*)
		Offset :	UDINT;(*Debug-Offset*)
		temp :	DWORD := DWORD#1;(*Debug-Offset*)
		MODE :	BOOL;(*modus*)
		faktor :	UDINT;(*Systemtakt-Faktor*)
		init :	BOOL;
		v_plc_ticks_per_sec :	UDINT;
		base :	UDINT := UDINT#1000;
	END_VAR

	IF init = FALSE THEN
		v_plc_ticks_per_sec := INT_TO_UDINT(PLC_TICKS_PER_SEC);
		IF v_plc_ticks_per_sec = UDINT#1024 THEN
			faktor := UDINT#1;
			MODE := FALSE;
		ELSIF v_plc_ticks_per_sec > UDINT#0 THEN
			IF v_plc_ticks_per_sec <= base THEN
				faktor := base / v_plc_ticks_per_sec;
				MODE := FALSE;
			ELSE
				faktor := v_plc_ticks_per_sec / base;
				MODE := TRUE;
			END_IF;
		ELSE
			faktor := UDINT#1;
		END_IF;
		init := TRUE;
	END_IF;

	IF MODE THEN
		T_PLC_MS := DINT_TO_UDINT(PLC_SYS_TICK_CNT) / faktor;
	ELSE
		T_PLC_MS := DINT_TO_UDINT(PLC_SYS_TICK_CNT) * faktor;
	END_IF;

	IF debug THEN
		T_PLC_MS := (DWORD_TO_UDINT(SHL(UDINT_TO_DWORD(T_PLC_MS),N) OR SHL(temp,N)) - UDINT#1) + Offset;
	END_IF;
END_FUNCTION_BLOCK

FUNCTION FRMP_B:BYTE
	VAR_INPUT
		START :	BYTE;
		DIR :	BOOL;
		TD :	TIME;
		TR :	TIME;
	END_VAR

	IF TD < TR THEN
		FRMP_B := MIN(UDINT_TO_BYTE(DWORD_TO_UDINT(SHL(TIME_TO_DWORD(TD), 8)) / TIME_TO_UDINT2(TR)), SEL(DIR, START, USINT_TO_BYTE(USINT#255 - BYTE_TO_USINT(START))));
		IF DIR THEN
			FRMP_B := USINT_TO_BYTE(BYTE_TO_USINT(START) + BYTE_TO_USINT(FRMP_B));
		ELSE
			FRMP_B := USINT_TO_BYTE(BYTE_TO_USINT(START) - BYTE_TO_USINT(FRMP_B));
		END_IF;
	ELSE
		FRMP_B := SEL(DIR, BYTE#0, BYTE#255);
	END_IF;
END_FUNCTION

FUNCTION_BLOCK _RMP_B
	VAR_INPUT
		DIR :	BOOL;
		E :	BOOL := TRUE;
		TR :	TIME;
	END_VAR

	VAR_IN_OUT
		RMP :	BYTE;
	END_VAR

	VAR
		T_PLC_MS :	T_PLC_MS_block;
		TX :	TIME;
		TL :	TIME;
		tn :	TIME;
		init :	BOOL;
		last_DIR :	BOOL;
		START :	BYTE;
	END_VAR

	T_PLC_MS();
	TX := UDINT_TO_TIME(T_PLC_MS.T_PLC_MS);

	IF E AND init AND (DIR = last_DIR) AND (RMP <> SEL(DIR, BYTE#0, BYTE#255)) AND TR = tn THEN
		RMP := FRMP_B(START, DIR, SUB_TIME(TX, TL), TR);
	ELSE
		init := TRUE;
		TL := TX;
		tn := tr;
		START := RMP;
	END_IF;
	last_DIR := DIR;
END_FUNCTION_BLOCK

FUNCTION_BLOCK RMP_B_Block

	VAR_INPUT
		SET :	BOOL;
		PT :	TIME;
		E :	BOOL := TRUE;
		UP :	BOOL := TRUE;
		RST :	BOOL;
	END_VAR

	VAR_OUTPUT
		OUT :	BYTE;
		BUSY :	BOOL;
		HIGH :	BOOL;
		LOW :	BOOL;
	END_VAR

	VAR
		rmp :	_RMP_B;
	END_VAR

	rmp(DIR := UP, E := E, TR := PT, RMP := OUT);
	OUT := rmp.RMP;

	IF RST THEN
		OUT := BYTE#0;
	ELSIF SET THEN
		OUT := BYTE#255;
	END_IF;

LOW := OUT = BYTE#0;
HIGH := OUT = BYTE#255;
busy := NOT (low OR high) AND E;

END_FUNCTION_BLOCK

FUNCTION_BLOCK BLIND_ACTUATOR_Block

	VAR_INPUT
		UP :	BOOL;
		DN :	BOOL;
		S_IN :	BYTE;
		T_UD :	TIME := T#10s;
		T_ANGLE :	TIME := T#3s;
		T_LOCKOUT :	TIME := t#100ms;
	END_VAR

	VAR_OUTPUT
		POS :	BYTE;
		ANG :	BYTE;
		QU :	BOOL;
		QD :	BOOL;
		STATUS :	BYTE;
	END_VAR

	VAR
		POSition :	RMP_B_Block;
		angle :	RMP_B_Block;
		lock :	INTERLOCK_Block;
	END_VAR

	lock(i1 := UP, I2 := DN, TL := T_lockOUT);

	angle(e := lock.Q1 OR lock.Q2, UP := lock.Q1, PT := T_Angle);
	POSition(e := lock.Q1 AND angle.high OR lock.Q2 AND angle.low, up := lock.Q1, PT := T_UD);

	POS := POSition.Out;
	ang := angle.Out;

	QU := lock.Q1;
	QD := lock.Q2;

	IF UP AND DN THEN
		STATUS := BYTE#1;
	ELSIF UP THEN
		STATUS := BYTE#121;
	ELSIF DN THEN
		IF DN THEN
		    STATUS := BYTE#1;
		ELSE
		    STATUS := BYTE#122;
		END_IF;
	ELSE
		STATUS := S_IN;
	END_IF;

END_FUNCTION_BLOCK

PROGRAM program0
	VAR
		UP :	BOOL;
		DN :	BOOL;
		S_IN :	BYTE;
		T_UD :	TIME := T#10s;
		T_ANGLE :	TIME := T#3s;
		T_LOCKOUT :	TIME := t#100ms;
		POS :	BYTE;
		ANG :	BYTE;
		QU :	BOOL;
		QD :	BOOL;
		func_block : BLIND_ACTUATOR_Block;
	END_VAR
	func_block.UP := UP;
	func_block.DN := DN;
	func_block.S_IN := S_IN ;
	func_block.T_UD := T_UD;
	func_block.T_ANGLE := T_ANGLE;
	func_block.T_LOCKOUT := T_LOCKOUT;
	func_block();
	POS  := func_block.POS;
	ANG  := func_block.ANG;
	QU  := func_block.QU;
	QD  := func_block.QD;
END_PROGRAM

(* ---- lb_claude_assisted_cf97dc740e86_0011.st ---- *)
(*
This code implements a randomly grown symbolic expression:

xor(xor(xor(xor(!((IN48 | (xor(xor(!(!(IN48)), !(!(xor(xor(IN15 & IN37, IN27 & IN43), xor(xor(IN10, IN50), IN49))))), !((IN7 & (xor(xor(IN34, IN29), IN41))) | ((IN34 & IN45) | (!(IN2))))))) & IN16), IN31), IN38), (IN16 | IN47) & IN28), (((!(IN20)) | ((xor(xor(xor(xor(((IN39 | IN35) | (IN9 & IN43)) & IN46, !((!(IN46)) | (xor(xor(IN5, IN34), IN46)))), (!(IN19 | IN49)) | (!(!(IN22)))), xor(xor(IN13, IN22), ((!(IN35)) & (xor(xor(IN2, IN40), IN38))) & IN43)), IN29)) | (xor(xor(!(!(xor(xor(IN8 | IN20, IN6 | IN40), xor(xor(IN12, IN18), IN33)))), !(((!(IN34)) & IN30) | ((!(IN31)) & (IN36 & IN6)))), (!(IN35)) & true)))) & ((((IN17 | (!(!(IN26 | IN42)))) | (xor(xor(IN44, ((xor(xor(IN13, IN3), IN47)) | (xor(xor(IN10, IN45), IN26))) & (xor(xor(!(IN3), IN34 | true), !(IN45)))), !(IN7 | IN35)))) & ((!(!(xor(xor(IN41 & IN25, xor(xor(IN10, IN9), IN48)), IN39)))) | (xor(xor(((xor(xor(IN22, IN35), IN30)) | (IN30 & IN45)) & ((IN24 | IN15) | IN48), !((xor(xor(IN16, IN5), IN23)) | (!(IN4)))), !((xor(xor(IN38, IN16), IN14)) | IN41))))) | ((IN27 & IN46) & ((xor(xor(!(!(xor(xor(IN29, IN24), IN24))), ((IN29 & IN32) & (IN36 | IN47)) | IN15), !(xor(xor(IN45, IN47 | IN29), xor(false, IN9))))) & (xor(xor(xor(xor((xor(xor(IN29, IN4), IN8)) & (!(IN27)), (xor(xor(IN24, IN23), IN10)) | IN19), (IN35 & IN15) | IN20), IN4 & ((!(IN9)) | (xor(xor(IN12, IN15), IN37)))), !(!(IN3)))))))) & (IN27 | IN9))

*)

FUNCTION_BLOCK F_CollectInput
  VAR_IN_OUT
      Data : ARRAY[1..50] OF BOOL;
  END_VAR
  VAR_INPUT
      TICK  : BOOL := 0;
      IN1   : BOOL := 0;
      IN2   : BOOL := 0;
      IN3   : BOOL := 0;
      IN4   : BOOL := 0;
      IN5   : BOOL := 0;
      RESET : BOOL := FALSE;
  END_VAR
  VAR_OUTPUT
      Finished : BOOL;
  END_VAR
  VAR
      j    : USINT := 1;
      tock : BOOL  := 0;
  END_VAR
  IF NOT RESET AND tock = NOT TICK THEN
      Data[j]   := IN1;
      Data[j+1] := IN2;
      Data[j+2] := IN3;
      Data[j+3] := IN4;
      Data[j+4] := IN5;
      j := j + 5;
      tock := TICK;
  ELSE
      j := 1;
      tock := 0;
  END_IF;
  Finished := (j > 50);
END_FUNCTION_BLOCK

PROGRAM Boiler
  VAR
    Data  : ARRAY[1..50] OF BOOL;
    Ready : BOOL;
    CollectInput : F_CollectInput;
  END_VAR
  VAR
    TICK     AT %IX1.0 : BOOL;
    IN1      AT %IX0.3 : BOOL;
    IN2      AT %IX0.4 : BOOL;
    IN3      AT %IX0.5 : BOOL;
    IN4      AT %IX0.6 : BOOL;
    IN5      AT %IX0.7 : BOOL;
    OutReady AT %QX0.0 : BOOL := FALSE;
    FeedNext AT %QX0.1 : BOOL := FALSE;
    Out      AT %QX0.2 : BOOL;
  END_VAR
  CollectInput(TICK:=TICK, IN1:=IN1, IN2:=IN2, IN3:=IN3, IN4:=IN4, IN5:=IN5);
  Ready := CollectInput.Finished;
  FeedNext := 1;
  IF Ready THEN
    Out := (((((NOT ((Data[48] OR (((NOT (NOT Data[48])) XOR (NOT (NOT (((Data[15] AND Data[37]) XOR (Data[27] AND Data[43])) XOR ((Data[10] XOR Data[50]) XOR Data[49]))))) XOR (NOT ((Data[7] AND ((Data[34] XOR Data[29]) XOR Data[41])) OR ((Data[34] AND Data[45]) OR (NOT Data[2])))))) AND Data[16])) XOR Data[31]) XOR Data[38]) XOR ((Data[16] OR Data[47]) AND Data[28])) XOR ((((NOT Data[20]) OR ((((((((Data[39] OR Data[35]) OR (Data[9] AND Data[43])) AND Data[46]) XOR (NOT ((NOT Data[46]) OR ((Data[5] XOR Data[34]) XOR Data[46])))) XOR ((NOT (Data[19] OR Data[49])) OR (NOT (NOT Data[22])))) XOR ((Data[13] XOR Data[22]) XOR (((NOT Data[35]) AND ((Data[2] XOR Data[40]) XOR Data[38])) AND Data[43]))) XOR Data[29]) OR (((NOT (NOT (((Data[8] OR Data[20]) XOR (Data[6] OR Data[40])) XOR ((Data[12] XOR Data[18]) XOR Data[33])))) XOR (NOT (((NOT Data[34]) AND Data[30]) OR ((NOT Data[31]) AND (Data[36] AND Data[6]))))) XOR ((NOT Data[35]) AND TRUE)))) AND ((((Data[17] OR (NOT (NOT (Data[26] OR Data[42])))) OR ((Data[44] XOR ((((Data[13] XOR Data[3]) XOR Data[47]) OR ((Data[10] XOR Data[45]) XOR Data[26])) AND (((NOT Data[3]) XOR (Data[34] OR TRUE)) XOR (NOT Data[45])))) XOR (NOT (Data[7] OR Data[35])))) AND ((NOT (NOT (((Data[41] AND Data[25]) XOR ((Data[10] XOR Data[9]) XOR Data[48])) XOR Data[39]))) OR ((((((Data[22] XOR Data[35]) XOR Data[30]) OR (Data[30] AND Data[45])) AND ((Data[24] OR Data[15]) OR Data[48])) XOR (NOT (((Data[16] XOR Data[5]) XOR Data[23]) OR (NOT Data[4])))) XOR (NOT (((Data[38] XOR Data[16]) XOR Data[14]) OR Data[41]))))) OR ((Data[27] AND Data[46]) AND ((((NOT (NOT ((Data[29] XOR Data[24]) XOR Data[24]))) XOR (((Data[29] AND Data[32]) AND (Data[36] OR Data[47])) OR Data[15])) XOR (NOT ((Data[45] XOR (Data[47] OR Data[29])) XOR (FALSE XOR Data[9])))) AND (((((((Data[29] XOR Data[4]) XOR Data[8]) AND (NOT Data[27])) XOR (((Data[24] XOR Data[23]) XOR Data[10]) OR Data[19])) XOR ((Data[35] AND Data[15]) OR Data[20])) XOR (Data[4] AND ((NOT Data[9]) OR ((Data[12] XOR Data[15]) XOR Data[37])))) XOR (NOT (NOT Data[3]))))))) AND (Data[27] OR Data[9])));
    IF Ready THEN
        OutReady := 0;
    ELSE
        OutReady := 1;
    END_IF;
    CollectInput(RESET:=TRUE);
  END_IF;
END_PROGRAM

CONFIGURATION Config0
  RESOURCE Res0 ON PLC
    TASK task0(INTERVAL := T#20ms,PRIORITY := 0);
    PROGRAM instance0 WITH task0 : Boiler;
  END_RESOURCE
END_CONFIGURATION

(* ---- lb_claude_assisted_cfaeee6d9c87_0028.st ---- *)
FUNCTION_BLOCK T_PLC_MS_block
	VAR_OUTPUT
		T_PLC_MS :	UDINT;
	END_VAR

	VAR_EXTERNAL
		PLC_TICKS_PER_SEC :	INT;
		PLC_SYS_TICK_CNT :	DINT;
	END_VAR

	VAR
		debug :	BOOL;(*Debug-Mode ON / OFF*)
		N :	INT;(*Debug-Faktor*)
		Offset :	UDINT;(*Debug-Offset*)
		temp :	DWORD := DWORD#1;(*Debug-Offset*)
		mode :	BOOL;(*modus*)
		faktor :	UDINT;(*Systemtakt-Faktor*)
		init :	BOOL;
		v_plc_ticks_per_sec :	UDINT;
		base :	UDINT := UDINT#1000;
	END_VAR

	IF init = FALSE THEN
		v_plc_ticks_per_sec := INT_TO_UDINT(PLC_TICKS_PER_SEC);
		IF v_plc_ticks_per_sec = UDINT#1024 THEN
			faktor := UDINT#1;
			mode := FALSE;
		ELSIF v_plc_ticks_per_sec > UDINT#0 THEN
			IF v_plc_ticks_per_sec <= base THEN
				faktor := base / v_plc_ticks_per_sec;
				mode := FALSE;
			ELSE
				faktor := v_plc_ticks_per_sec / base;
				IF v_plc_ticks_per_sec > UDINT#0 THEN
				    mode := FALSE;
				ELSE
				    mode := TRUE;
				END_IF;
			END_IF;
		ELSE
			faktor := UDINT#1;
		END_IF;
		init := TRUE;
	END_IF;

	IF mode THEN
		T_PLC_MS := DINT_TO_UDINT(PLC_SYS_TICK_CNT) / faktor;
	ELSE
		T_PLC_MS := DINT_TO_UDINT(PLC_SYS_TICK_CNT) * faktor;
	END_IF;

	IF debug THEN
		T_PLC_MS := (DWORD_TO_UDINT(SHL(UDINT_TO_DWORD(T_PLC_MS),N) OR SHL(temp,N)) - UDINT#1) + Offset;
	END_IF;
END_FUNCTION_BLOCK

FUNCTION_BLOCK M_TX_Block

	VAR_INPUT
		IN :	BOOL;
		TMAX :	TIME := t#10d;
		RST :	BOOL;
	END_VAR

	VAR_OUTPUT
		TH :	TIME;
		TL :	TIME;
		DC :	REAL;
		F :	REAL;
		ET :	TIME;
	END_VAR

	VAR
		edge :	BOOL;
		start :	TIME;
		stop :	TIME;
		tx :	TIME;
		rise :	BOOL;
		fall :	BOOL;
		startup :	BOOL;
		T_PLC_MS :	T_PLC_MS_block;
	END_VAR

	IF rst OR (et >= tmax) THEN
		rise := FALSE;
		fall := FALSE;
		startup := FALSE;
		th := t#0ms;
		tl := t#0ms;
		DC := 0.0;
		F := 0.0;
		ET := t#0s;
	END_IF;

	(* avoid timers to start when input is true at startup *)
	IF NOT startup THEN
		edge := in;
		startup := TRUE;
	END_IF;

	(* read system timer *)
	T_PLC_MS();
	tx:= UDINT_TO_TIME(T_PLC_MS.T_PLC_MS);

	(* edge trigger rising and falling edge *)
	IF in XOR edge THEN
		edge := in;
		(* rising edge starts measurement *)
		IF in THEN
			start := Tx;
			rise := TRUE;
			IF fall THEN tl := start - stop; END_IF;
			IF th > t#0ms AND tl > t#0ms THEN
				dc := TIME_TO_REAL(th) / TIME_TO_REAL(th+tl);
				f := 1000.0 / TIME_TO_REAL(th + tl);
			END_IF;
		(* falling edge starts second cycle measurement *)
		ELSE
			stop := Tx;
			fall := TRUE;
			IF rise THEN th := stop - start; END_IF;
			IF th > t#0ms AND tl > t#0ms THEN
				dc := TIME_TO_REAL(th) /  TIME_TO_REAL(th+tl);
				f := 1000.0 / TIME_TO_REAL(th + tl);
			END_IF;
		END_IF;
	END_IF;
	IF rise THEN et := tx - start; END_IF;

	(* check FOR rst input *)
	IF rst OR (et >= tmax) THEN
		rise := FALSE;
		fall := FALSE;
		startup := FALSE;
		th := t#0ms;
		tl := t#0ms;
		DC := 0.0;
		F := 0.0;
		ET := t#0s;
	END_IF;

	(* avoid timers to start when input is true at startup *)
	IF NOT startup THEN
		edge := in;
		startup := TRUE;
	END_IF;

	(* read system timer *)
	T_PLC_MS();
	tx:= UDINT_TO_TIME(T_PLC_MS.T_PLC_MS);

	(* edge trigger rising and falling edge *)
	IF in XOR edge THEN
		edge := in;
		(* rising edge starts measurement *)
		IF in THEN
			start := Tx;
			rise := TRUE;
			IF fall THEN tl := start - stop; END_IF;
			IF th > t#0ms AND tl > t#0ms THEN
				dc := TIME_TO_REAL(th) / TIME_TO_REAL(th+tl);
				f := 1000.0 / TIME_TO_REAL(th + tl);
			END_IF;
		(* falling edge starts second cycle measurement *)
		ELSE
			stop := Tx;
			fall := TRUE;
			IF rise THEN th := stop - start; END_IF;
			IF th > t#0ms AND tl > t#0ms THEN
				dc := TIME_TO_REAL(th) /  TIME_TO_REAL(th+tl);
				f := 1000.0 / TIME_TO_REAL(th + tl);
			END_IF;
		END_IF;
	END_IF;
	IF rise THEN et := tx - start; END_IF;

END_FUNCTION_BLOCK

PROGRAM program0

	VAR
		IN :	BOOL;
		TMAX :	TIME := t#10d;
		RST :	BOOL;

		TH :	TIME;
		TL :	TIME;
		DC :	REAL;
		F :	REAL;
		ET :	TIME;

		func_block : M_TX_Block;
	END_VAR
	func_block.IN := IN;
	func_block.TMAX := TMAX;
	func_block.RST := RST;

	func_block();
	TH := func_block.TH;
	TL := func_block.TL;
	DC := func_block.DC;
	F := func_block.F;
	ET := func_block.ET;

END_PROGRAM

CONFIGURATION Config0

	VAR_GLOBAL
		PLC_TICKS_PER_SEC :	INT;
		PLC_SYS_TICK_CNT :	DINT;
	END_VAR

	RESOURCE Res0 ON PLC
		TASK task0(INTERVAL := T#20ms,PRIORITY := 0);
		PROGRAM instance0 WITH task0 : program0;
	END_RESOURCE

END_CONFIGURATION

(* ---- lb_claude_assisted_d057941c9efc_0056.st ---- *)
(*
This code implements a randomly grown symbolic expression:

(!((!(IN3)) & ((((!(xor(xor(xor(xor(xor(xor(IN22, IN40), IN38), !(IN44)), IN20), IN22), xor(xor(!(IN6), true & IN32), !(IN17))))) | IN31) | (IN3 | IN14)) | IN48))) | ((((!(IN45 & (((xor(xor(IN37 & IN23, IN35), IN11 & IN15)) & IN46) | ((!(IN28 | IN33)) | (!(!(IN13))))))) & IN19) & ((((xor(xor(IN22, !(!(IN40 & IN38))), (xor(xor(IN11 & IN33, IN46 | IN15), IN35 & IN15)) | (!(IN15 | IN17)))) & (!(((IN2 & IN17) | (!(IN16))) & IN16))) & (IN40 | IN25)) & true)) | (xor(xor(IN40, IN11), IN10)))

*)

FUNCTION_BLOCK F_CollectInput
  VAR_IN_OUT
      Data : ARRAY[1..50] OF BOOL;
  END_VAR
  VAR_INPUT
      TICK  : BOOL := 0;
      IN1   : BOOL := 0;
      IN2   : BOOL := 0;
      IN3   : BOOL := 0;
      IN4   : BOOL := 0;
      IN5   : BOOL := 0;
      RESET : BOOL := FALSE;
  END_VAR
  VAR_OUTPUT
      Finished : BOOL;
  END_VAR
  VAR
      j    : USINT := 1;
      tock : BOOL  := 0;
  END_VAR
  IF NOT RESET AND tock = NOT TICK THEN
      Data[j]   := IN1;
      Data[j+1] := IN2;
      Data[j+2] := IN3;
      Data[j+3] := IN4;
      Data[j+4] := IN5;
      j := j + 5;
      tock := TICK;
  ELSE
      j := 1;
      tock := 0;
  END_IF;
  Finished := (j > 50);
END_FUNCTION_BLOCK

PROGRAM Boiler
  VAR
    Data  : ARRAY[1..50] OF BOOL;
    Ready : BOOL;
    CollectInput : F_CollectInput;
  END_VAR
  VAR
    TICK     AT %IX1.0 : BOOL;
    IN1      AT %IX0.3 : BOOL;
    IN2      AT %IX0.4 : BOOL;
    IN3      AT %IX0.5 : BOOL;
    IN4      AT %IX0.6 : BOOL;
    IN5      AT %IX0.7 : BOOL;
    OutReady AT %QX0.0 : BOOL := FALSE;
    FeedNext AT %QX0.1 : BOOL := FALSE;
    Out      AT %QX0.2 : BOOL;
  END_VAR
  CollectInput(TICK:=TICK, IN1:=IN1, IN2:=IN2, IN3:=IN3, IN4:=IN4, IN5:=IN5);
  Ready := CollectInput.Finished;
  FeedNext := 1;
  IF Ready THEN
    Out := ((NOT ((NOT Data[3]) AND ((((NOT ((((((Data[22] XOR Data[40]) XOR Data[38]) XOR (NOT Data[44])) XOR Data[20]) XOR Data[22]) XOR (((NOT Data[6]) XOR (TRUE AND Data[32])) XOR (NOT Data[17])))) OR Data[31]) OR (Data[3] OR Data[14])) OR Data[48]))) OR ((((NOT (Data[45] AND (((((Data[37] AND Data[23]) XOR Data[35]) XOR (Data[11] AND Data[15])) AND Data[46]) OR ((NOT (Data[28] OR Data[33])) OR (NOT (NOT Data[13])))))) AND Data[19]) AND (((((Data[22] XOR (NOT (NOT (Data[40] AND Data[38])))) XOR ((((Data[11] AND Data[33]) XOR (Data[46] OR Data[15])) XOR (Data[35] AND Data[15])) OR (NOT (Data[15] OR Data[17])))) AND (NOT (((Data[2] AND Data[17]) OR (NOT Data[16])) AND Data[16]))) AND (Data[40] OR Data[25])) AND TRUE)) OR ((Data[40] XOR Data[11]) XOR Data[10])));
    IF Ready THEN
        OutReady := 0;
    ELSE
        OutReady := 1;
    END_IF;
    CollectInput(RESET:=TRUE);
  END_IF;
END_PROGRAM

CONFIGURATION Config0
  RESOURCE Res0 ON PLC
    TASK task0(INTERVAL := T#20ms,PRIORITY := 0);
    PROGRAM instance0 WITH task0 : Boiler;
  END_RESOURCE
END_CONFIGURATION

(* ---- lb_claude_assisted_d05b3fabb5c2_0024.st ---- *)
(*
This code implements a randomly grown symbolic expression:

(!(IN26 & (IN45 | ((xor(xor(IN3, !(xor(xor((IN43 & IN34) | (IN19 | IN26), xor(xor(!(IN50), IN21 | IN1), IN17 & IN23)), xor(xor(xor(xor(IN4, IN2), IN41), IN7 & IN29), IN13)))), IN42)) | IN20)))) | (!((xor(xor(!(!(xor(xor(!((!(IN14)) & IN36), ((xor(xor(IN45, IN34), IN41)) | (IN17 | IN11)) & IN16), !(xor(xor(IN37 & IN25, true), IN17 & IN22))))), !((!(IN31)) | (!(IN6)))), ((!(IN16)) | IN27) & (IN46 & ((xor(xor(!(IN15 | IN34), IN28), !(IN7 & IN3))) & ((xor(xor(!(IN32), xor(xor(IN36, IN43), IN28)), !(IN36))) & IN44))))) & IN13))

*)

FUNCTION_BLOCK F_CollectInput
  VAR_IN_OUT
      Data : ARRAY[1..50] OF BOOL;
  END_VAR
  VAR_INPUT
      TICK  : BOOL := 0;
      IN1   : BOOL := 0;
      IN2   : BOOL := 0;
      IN3   : BOOL := 0;
      IN4   : BOOL := 0;
      IN5   : BOOL := 0;
      RESET : BOOL := FALSE;
  END_VAR
  VAR_OUTPUT
      Finished : BOOL;
  END_VAR
  VAR
      j    : USINT := 1;
      tock : BOOL  := 0;
  END_VAR
  IF NOT RESET AND tock = NOT TICK THEN
      Data[j]   := IN1;
      Data[j+1] := IN2;
      Data[j+2] := IN3;
      Data[j+3] := IN4;
      Data[j+4] := IN5;
      j := j + 5;
      tock := TICK;
  ELSE
      j := 1;
      tock := 0;
  END_IF;
  Finished := (j > 50);
END_FUNCTION_BLOCK

PROGRAM Boiler
  VAR
    Data  : ARRAY[1..50] OF BOOL;
    Ready : BOOL;
    CollectInput : F_CollectInput;
  END_VAR
  VAR
    TICK     AT %IX1.0 : BOOL;
    IN1      AT %IX0.3 : BOOL;
    IN2      AT %IX0.4 : BOOL;
    IN3      AT %IX0.5 : BOOL;
    IN4      AT %IX0.6 : BOOL;
    IN5      AT %IX0.7 : BOOL;
    OutReady AT %QX0.0 : BOOL := FALSE;
    FeedNext AT %QX0.1 : BOOL := FALSE;
    Out      AT %QX0.2 : BOOL;
  END_VAR
  CollectInput(TICK:=TICK, IN1:=IN1, IN2:=IN2, IN3:=IN3, IN4:=IN4, IN5:=IN5);
  Ready := CollectInput.Finished;
  FeedNext := 1;
  IF Ready THEN
    Out := ((NOT (Data[26] AND (Data[45] OR (((Data[3] XOR (NOT ((((Data[43] AND Data[34]) OR (Data[19] OR Data[26])) XOR (((NOT Data[50]) XOR (Data[21] OR Data[1])) XOR (Data[17] AND Data[23]))) XOR ((((Data[4] XOR Data[2]) XOR Data[41]) XOR (Data[7] AND Data[29])) XOR Data[13])))) XOR Data[42]) OR Data[20])))) OR (NOT ((((NOT (NOT (((NOT ((NOT Data[14]) AND Data[36])) XOR ((((Data[45] XOR Data[34]) XOR Data[41]) OR (Data[17] OR Data[11])) AND Data[16])) XOR (NOT (((Data[37] AND Data[25]) XOR TRUE) XOR (Data[17] AND Data[22])))))) XOR (NOT ((NOT Data[31]) OR (NOT Data[6])))) XOR (((NOT Data[16]) OR Data[27]) AND (Data[46] AND ((((NOT (Data[15] OR Data[34])) XOR Data[28]) XOR (NOT (Data[7] AND Data[3]))) AND ((((NOT Data[32]) XOR ((Data[36] XOR Data[43]) XOR Data[28])) XOR (NOT Data[36])) AND Data[44]))))) AND Data[13])));
    IF Ready THEN
        OutReady := 0;
    ELSE
        OutReady := 1;
    END_IF;
    CollectInput(RESET:=TRUE);
  END_IF;
END_PROGRAM

CONFIGURATION Config0
  RESOURCE Res0 ON PLC
    TASK task0(INTERVAL := T#20ms,PRIORITY := 0);
    PROGRAM instance0 WITH task0 : Boiler;
  END_RESOURCE
END_CONFIGURATION

(* ---- lb_claude_assisted_d14a62c1c3ac_0110.st ---- *)
FUNCTION _REAL_TO_UDINT:UDINT
  VAR_INPUT
    X :	REAL;
  END_VAR

  IF REAL_TO_UDINT(0.5) = UDINT#1 THEN
    _REAL_TO_UDINT := REAL_TO_UDINT(X);
  ELSIF X > 0.0 THEN
    _REAL_TO_UDINT := REAL_TO_UDINT(X+0.5);
  ELSIF X < 0.0 THEN
    _REAL_TO_UDINT := REAL_TO_UDINT(X-0.5);
  ELSE
    _REAL_TO_UDINT := UDINT#0;
  END_IF;
END_FUNCTION

FUNCTION REAL_TO_TIME2:TIME
	VAR_INPUT
		IN :	REAL;
	END_VAR

	REAL_TO_TIME2 := DINT_TO_TIME(UDINT_TO_DINT(_REAL_TO_UDINT(IN)));
END_FUNCTION

FUNCTION_BLOCK T_PLC_US_Block
	VAR_OUTPUT
		T_PLC_US :	UDINT;
	END_VAR

	VAR
		PLC_TICKS_PER_SEC :	INT;
		PLC_SYS_TICK_CNT :	DINT;
	END_VAR

	VAR
		debug :	BOOL;
		N :	INT;
		Offset :	UDINT;
		temp :	DWORD := DWORD#1;
		MODE :	BOOL;
		faktor :	UDINT;
		init :	BOOL;
		v_plc_ticks_per_sec :	UDINT;
		base :	UDINT := UDINT#1000000;
	END_VAR

	IF init = FALSE THEN
		v_plc_ticks_per_sec := INT_TO_UDINT(PLC_TICKS_PER_SEC);
		IF v_plc_ticks_per_sec = UDINT#1024 THEN
			faktor := UDINT#1000;
			MODE := FALSE;
		ELSIF v_plc_ticks_per_sec > UDINT#0 THEN
			IF v_plc_ticks_per_sec <= base THEN
				faktor := base / v_plc_ticks_per_sec;
				MODE := FALSE;
			ELSE
				faktor := v_plc_ticks_per_sec / base;
				MODE := TRUE;
			END_IF;
		ELSE
			faktor := UDINT#1;
		END_IF;
		init := TRUE;
	END_IF;

	IF MODE THEN
		T_PLC_US := DINT_TO_UDINT(PLC_SYS_TICK_CNT) / faktor;
	ELSE
		T_PLC_US := DINT_TO_UDINT(PLC_SYS_TICK_CNT) * faktor;
	END_IF;

	IF debug THEN
		T_PLC_US := (DWORD_TO_UDINT(SHL(UDINT_TO_DWORD(T_PLC_US),N) OR SHL(temp,N)) - UDINT#1) + Offset;
	END_IF;
END_FUNCTION_BLOCK

FUNCTION_BLOCK FT_DERIV
	VAR_INPUT
		IN :	REAL;
		K :	REAL := 1.0;
		RUN :	BOOL := TRUE;
	END_VAR

	VAR_OUTPUT
		OUT :	REAL;
	END_VAR

	VAR
		old :	REAL;
		TX :	UDINT;
		last :	UDINT;
		init :	BOOL;
		tc :	REAL;
		T_PLC_US :	T_PLC_US_Block;
	END_VAR

	T_PLC_US();
	TX:= T_PLC_US.T_PLC_US;
	tc := UDINT_TO_REAL(TX - last);

	IF NOT init THEN
		init := TRUE;
		old := IN;
	ELSIF RUN AND tc > 0.0 THEN
		OUT := (IN - old) / tc * 1000000.0 * K;
		old := IN;
	ELSE
		OUT := 0.0;
	END_IF;

	last := TX;

	T_PLC_US();
	TX:= T_PLC_US.T_PLC_US;

	IF NOT init THEN
		init := TRUE;
	ELSIF RUN AND (TX - last) > UDINT#0 THEN
		OUT := (IN - old) / UDINT_TO_REAL(TX - last) * 1000000.0 * K;
	ELSE
		OUT := 0.0;
	END_IF;
	old := IN;
	last := TX;
END_FUNCTION_BLOCK

FUNCTION_BLOCK FT_PT1

	VAR_INPUT
		IN :	REAL;
		T :	TIME;
		K :	REAL := 1.0;
	END_VAR

	VAR_OUTPUT
		OUT :	REAL;
	END_VAR

	VAR
		last :	UDINT;
		TX :	UDINT;
		init :	BOOL;
		T_PLC_US :	T_PLC_US_Block;
	END_VAR

	T_PLC_US();
	TX:= T_PLC_US.T_PLC_US;

	IF NOT init OR T = t#0s THEN
		init := TRUE;
		OUT := K * IN;
	ELSE
		IF NOT init OR T = t#0s THEN
		    OUT := K * IN;
		ELSE
		    OUT := OUT + (IN * K - OUT) * UDINT_TO_REAL(TX - last) / TIME_TO_REAL(T) * 1.0E-3;
		END_IF;
		IF ABS(OUT) < 1.0E-20 THEN OUT := 0.0; END_IF;
	END_IF;
	last := TX;
END_FUNCTION_BLOCK

FUNCTION_BLOCK FT_PDT1_Block

	VAR_INPUT
		IN :	REAL;
		KP :	REAL := 1.0;
		TV :	REAL := 1.0;
		T1 :	REAL := 1.0;
	END_VAR

	VAR_OUTPUT
		Y :	REAL;
	END_VAR

	VAR
		diff :	FT_DERIV;
		_TP :	FT_PT1;
	END_VAR

	diff(IN := IN, K := TV);

	_TP(IN := diff.OUT, T := REAL_TO_TIME2(T1));

	Y := KP * (_TP.OUT + IN);

END_FUNCTION_BLOCK

PROGRAM program0
	VAR
		IN :	REAL;
		KP :	REAL := 1.0;
		TV :	REAL := 1.0;
		T1 :	REAL := 1.0;

		Y :	REAL;
		func_block : FT_PDT1_Block;
	END_VAR
	func_block.IN :=IN;
	func_block.KP :=KP;
	func_block.TV :=TV;
	func_block.T1 :=T1;
	func_block();
	Y := func_block.Y;
END_PROGRAM

(* ---- lb_claude_assisted_d275cc03958d_0091.st ---- *)
FUNCTION D_TRUNC : DINT
  VAR_INPUT
    x : REAL;
  END_VAR

  D_TRUNC := REAL_TO_DINT(X);
  IF X > 0.0 THEN
  	IF DINT_TO_REAL(D_TRUNC) > X THEN D_TRUNC := D_TRUNC - DINT#1; END_IF;
  ELSE
  	IF DINT_TO_REAL(D_TRUNC) < X THEN D_TRUNC := D_TRUNC + DINT#1; END_IF;
  END_IF;
END_FUNCTION

FUNCTION BIT_COUNT:INT

	VAR_INPUT
		IN :	DWORD;
	END_VAR

	VAR
		in_temp :	DWORD;
	END_VAR

	in_temp := IN;
	WHILE in_temp > DWORD#0 DO
		IF (in_temp AND DWORD#16#00000001) > DWORD#0 THEN Bit_Count := Bit_Count +1; END_IF;
		in_temp := SHR(in_temp,1);
	END_WHILE;

END_FUNCTION

FUNCTION FRACT:REAL
	VAR_INPUT
		X :	REAL;
	END_VAR

	IF ABS(x) < 2.0E9 THEN
		FRACT := x - DINT_TO_REAL(D_TRUNC(x));
	ELSE
		FRACT := 0.0;
	END_IF;

END_FUNCTION

FUNCTION_BLOCK T_PLC_MS_block
	VAR_OUTPUT
		T_PLC_MS :	UDINT;
	END_VAR

	VAR_EXTERNAL
		PLC_TICKS_PER_SEC :	INT;
		PLC_SYS_TICK_CNT :	DINT;
	END_VAR

	VAR
		debug :	BOOL;(*Debug-Mode ON / OFF*)
		N :	INT;(*Debug-Faktor*)
		Offset :	UDINT;(*Debug-Offset*)
		temp :	DWORD := DWORD#1;(*Debug-Offset*)
		mode :	BOOL;(*modus*)
		faktor :	UDINT;(*Systemtakt-Faktor*)
		init :	BOOL;
		v_plc_ticks_per_sec :	UDINT;
		base :	UDINT := UDINT#1000;
	END_VAR

	IF init = FALSE THEN
		v_plc_ticks_per_sec := INT_TO_UDINT(PLC_TICKS_PER_SEC);
		IF v_plc_ticks_per_sec = UDINT#1024 THEN
			faktor := UDINT#1;
			mode := FALSE;
		ELSIF v_plc_ticks_per_sec > UDINT#0 THEN
			IF v_plc_ticks_per_sec <= base THEN
				faktor := base / v_plc_ticks_per_sec;
				mode := FALSE;
			ELSE
				faktor := v_plc_ticks_per_sec / base;
				mode := TRUE;
			END_IF;
		ELSE
			faktor := UDINT#1;
		END_IF;
		init := TRUE;
	END_IF;

	IF mode THEN
		T_PLC_MS := DINT_TO_UDINT(PLC_SYS_TICK_CNT) / faktor;
	ELSE
		IF mode THEN
		    T_PLC_MS := DINT_TO_UDINT(PLC_SYS_TICK_CNT) / faktor;
		ELSE
		    T_PLC_MS := DINT_TO_UDINT(PLC_SYS_TICK_CNT) * faktor;
		END_IF;
	END_IF;

	IF debug THEN
		T_PLC_MS := (DWORD_TO_UDINT(SHL(UDINT_TO_DWORD(T_PLC_MS),N) OR SHL(temp,N)) - UDINT#1) + Offset;
	END_IF;

END_FUNCTION_BLOCK

FUNCTION BIT_LOAD_DW:DWORD

	VAR_INPUT
		IN :	DWORD;
		VAL :	BOOL;
		POS :	INT;
	END_VAR

	IF val THEN
		BIT_LOAD_DW := in OR SHL(DWORD#1,pos);
	ELSE
		BIT_LOAD_DW := in AND (NOT SHL(DWORD#1,pos));
	END_IF;

END_FUNCTION

FUNCTION BIT_OF_DWORD : BOOL
  VAR_INPUT
    IN : DWORD;
    N : INT;
  END_VAR

  BIT_OF_DWORD := (SHR(in,N) AND 16#00000001) > 0;
  (* from OSCAT library; www.oscat.de  *)
END_FUNCTION

FUNCTION _INT_TO_UDINT:UDINT
	VAR_INPUT
		IN :	INT;
	END_VAR

	_INT_TO_UDINT := DINT_TO_UDINT(INT_TO_DINT(IN));
END_FUNCTION

FUNCTION _DWORD_TO_REAL:REAL
	VAR_INPUT
		IN :	DWORD;
	END_VAR

	_DWORD_TO_REAL := UDINT_TO_REAL(DWORD_TO_UDINT(IN));

END_FUNCTION

FUNCTION_BLOCK RDM_block
	VAR_INPUT
		LAST :	REAL;
	END_VAR
	VAR_OUTPUT
		RDM :	REAL;
	END_VAR
	VAR
		T_PLC_MS :	T_PLC_MS_block;
		tn :	DWORD;
		tc :	INT;
	END_VAR
	T_PLC_MS();
	tn := UDINT_TO_DWORD(T_PLC_MS.T_PLC_MS);
	tc := Bit_Count(tn);

	tn:=BIT_LOAD_DW(tn,BIT_OF_DWORD(tn,2),31); (* tn.31 := tn.2; *)
	tn:=BIT_LOAD_DW(tn,BIT_OF_DWORD(tn,5),30); (* tn.30 := tn.5; *)
	tn:=BIT_LOAD_DW(tn,BIT_OF_DWORD(tn,4),29); (* tn.29 := tn.4; *)
	tn:=BIT_LOAD_DW(tn,BIT_OF_DWORD(tn,1),28); (* tn.28 := tn.1; *)
	tn:=BIT_LOAD_DW(tn,BIT_OF_DWORD(tn,0),27); (* tn.27 := tn.0; *)
	tn:=BIT_LOAD_DW(tn,BIT_OF_DWORD(tn,7),26); (* tn.26 := tn.7; *)
	tn:=BIT_LOAD_DW(tn,BIT_OF_DWORD(tn,6),25); (* tn.25 := tn.6; *)
	tn:=BIT_LOAD_DW(tn,BIT_OF_DWORD(tn,3),24); (* tn.24 := tn.3; *)

	tn := ROL(tn,Bit_Count(tn)) OR DWORD#16#80000001;
	tn := UDINT_TO_DWORD(DWORD_TO_UDINT(tn) MOD UDINT#71474513 + _INT_TO_UDINT(tc) + UDINT#77);
	RDM := fract(_DWORD_TO_REAL(tn) / 10000000.0 * (2.71828182845904523536028747135266249 - LIMIT_REAL(0.0,last,1.0)));
END_FUNCTION_BLOCK

FUNCTION_BLOCK GEN_RDM_Block

	VAR_INPUT
		PT :	TIME;
		AM :	REAL := REAL#1.0;
		OS :	REAL;
	END_VAR

	VAR_OUTPUT
		Q :	BOOL;
		Out :	REAL;
	END_VAR

	VAR
		tx :	TIME;
		last :	TIME;
		init :	BOOL;
		T_PLC_MS :	T_PLC_MS_Block;
		FB_rdm :	RDM_block;
	END_VAR

	T_PLC_MS();
	tx:= UDINT_TO_TIME(T_PLC_MS.T_PLC_MS) - last;

	IF NOT init THEN
		init := TRUE;
		last := tx;
		tx := t#0s;
	END_IF;

	IF tx >= pt THEN
		last := last + pt;
		tx := tx - pt;

		FB_rdm(last:=0.0);
		out := am * (FB_rdm.RDM - 0.5) + os;
		q := TRUE;
	ELSE
		q := FALSE;
	END_IF;

END_FUNCTION_BLOCK

PROGRAM program0
  VAR
	PT :	TIME;
	AM :	REAL := REAL#1.0;
	OS :	REAL;
	Q :	BOOL;
	Out :	REAL;
	func_block : GEN_RDM_Block;
  END_VAR
	func_block.PT  :=PT;
	func_block.AM  :=AM;
	func_block.OS  :=OS;
	func_block();
	Q := func_block.Q;
	Out := func_block.Out;
END_PROGRAM

CONFIGURATION Config0
	VAR_GLOBAL
		PLC_TICKS_PER_SEC :	INT;
		PLC_SYS_TICK_CNT :	DINT;
	END_VAR
	RESOURCE Res0 ON PLC
		TASK task0(INTERVAL := T#20ms,PRIORITY := 0);
		PROGRAM instance0 WITH task0 : program0;
	END_RESOURCE
END_CONFIGURATION

(* ---- lb_claude_assisted_d55caa1b42b9_0106.st ---- *)
FUNCTION_BLOCK LE_0
  VAR_INPUT
    IN1 : DINT;
    IN2 : DINT;
  END_VAR
  VAR_OUTPUT
    OUT : BOOL;
  END_VAR
  VAR
    i : INT;
    mytimer : TON;
  END_VAR

  OUT:=FALSE;
  IF IN1<=IN2 then
    OUT:=TRUE;
  END_IF;
  IF mytimer.Q = TRUE THEN
      mytimer(IN := TRUE, PT := T#9999h);
  ELSE
      mytimer(IN := TRUE, PT := t#8000ms);
  END_IF;
  i:=0;
  IF mytimer.Q = TRUE then
     WHILE i<4 do
      OUT:=TRUE;
    End_WHILE;
  End_IF;
END_FUNCTION_BLOCK

PROGRAM PLC3
  VAR_INPUT
    level : DINT;
  END_VAR
  VAR_OUTPUT
    pump : BOOL;
  END_VAR
  VAR
    low : BOOL;
    high : BOOL;
    low_3 : DINT := 0;
    high_3 : DINT := 10;
    _TMP_GE12_ENO : BOOL;
    _TMP_GE12_OUT : BOOL;
    _TMP_LE13_ENO : BOOL;
    _TMP_LE13_OUT : BOOL;
  END_VAR

  _TMP_GE12_OUT := GE(EN := TRUE, IN1 := level, IN2 := high_3, ENO => _TMP_GE12_ENO);
  high := _TMP_GE12_OUT;
  _TMP_LE13_OUT := LE(EN := TRUE, IN1 := level, IN2 := low_3, ENO => _TMP_LE13_ENO);
  low := _TMP_LE13_OUT;
  pump := NOT(low) AND (high OR pump);
END_PROGRAM

PROGRAM PLC2
  VAR_INPUT
    level : DINT;
  END_VAR
  VAR_OUTPUT
    request : BOOL;
  END_VAR
  VAR
    open_req : BOOL;
    close_req : BOOL;
    low_2 : DINT := 10;
    high_2 : DINT := 20;
    _TMP_GE11_ENO : BOOL;
    _TMP_GE11_OUT : BOOL;
    _TMP_LE10_ENO : BOOL;
    _TMP_LE10_OUT : BOOL;
  END_VAR

  _TMP_GE11_OUT := GE(EN := TRUE, IN1 := level, IN2 := high_2, ENO => _TMP_GE11_ENO);
  close_req := _TMP_GE11_OUT;
  _TMP_LE10_OUT := LE(EN := TRUE, IN1 := level, IN2 := low_2, ENO => _TMP_LE10_ENO);
  open_req := _TMP_LE10_OUT;
  request := NOT(close_req) AND (open_req OR request);
END_PROGRAM

PROGRAM PLC1
  VAR_INPUT
    level : DINT;
    request : DINT;
  END_VAR
  VAR_OUTPUT
    pumps : BOOL;
    valve : BOOL;
  END_VAR
  VAR
    low : BOOL;
    high : BOOL;
    open_req : BOOL;
    close_req : BOOL;
    low_1 : DINT := 40;
    high_1 : DINT := 80;
    LE_00 : LE_0;
    _TMP_GE33_ENO : BOOL;
    _TMP_GE33_OUT : BOOL;
    _TMP_EQ31_ENO : BOOL;
    _TMP_EQ31_OUT : BOOL;
    _TMP_EQ24_ENO : BOOL;
    _TMP_EQ24_OUT : BOOL;
  END_VAR

  LE_00(EN := TRUE, IN1 := level, IN2 := low_1);
  low := LE_00.OUT;
  _TMP_GE33_OUT := GE(EN := TRUE, IN1 := level, IN2 := high_1, ENO => _TMP_GE33_ENO);
  high := _TMP_GE33_OUT;
  pumps := NOT(high) AND (low OR pumps);
  valve := NOT(close_req) AND (valve OR open_req AND NOT(low));
  _TMP_EQ31_OUT := EQ(EN := TRUE, IN1 := request, IN2 := 1, ENO => _TMP_EQ31_ENO);
  open_req := _TMP_EQ31_OUT;
  _TMP_EQ24_OUT := EQ(EN := TRUE, IN1 := request, IN2 := 0, ENO => _TMP_EQ24_ENO);
  close_req := _TMP_EQ24_OUT;
END_PROGRAM

CONFIGURATION Config0

  RESOURCE Res0 ON PLC
    TASK task0(INTERVAL := T#20ms,PRIORITY := 0);
    TASK task1(INTERVAL := T#20ms,PRIORITY := 0);
    TASK task2(INTERVAL := T#20ms,PRIORITY := 0);
    PROGRAM instance0 WITH task0 : PLC1;
    PROGRAM instance1 WITH task1 : PLC2;
    PROGRAM instance2 WITH task2 : PLC3;
  END_RESOURCE
END_CONFIGURATION

(* ---- lb_claude_assisted_d5e23eaffa72_0034.st ---- *)
FUNCTION UDINT_TO_TIME2:TIME

	VAR_INPUT
		IN :	UDINT;
	END_VAR

	UDINT_TO_TIME2 := DINT_TO_TIME(UDINT_TO_DINT(IN));

END_FUNCTION

FUNCTION_BLOCK T_PLC_MS_block
	VAR_OUTPUT
		T_PLC_MS :	UDINT;
	END_VAR

	VAR
		PLC_TICKS_PER_SEC :	INT;
		PLC_SYS_TICK_CNT :	DINT;
	END_VAR

	VAR
		debug :	BOOL;(*Debug-Mode ON / OFF*)
		N :	INT;(*Debug-Faktor*)
		Offset :	UDINT;(*Debug-Offset*)
		temp :	DWORD := DWORD#1;(*Debug-Offset*)
		MODE :	BOOL;(*modus*)
		faktor :	UDINT;(*Systemtakt-Faktor*)
		init :	BOOL;
		v_plc_ticks_per_sec :	UDINT;
		base :	UDINT := UDINT#1000;
	END_VAR

	IF init = FALSE THEN
		v_plc_ticks_per_sec := INT_TO_UDINT(PLC_TICKS_PER_SEC);
		IF v_plc_ticks_per_sec = UDINT#1024 THEN
			faktor := UDINT#1;
			MODE := FALSE;
		ELSIF v_plc_ticks_per_sec > UDINT#0 THEN
			IF v_plc_ticks_per_sec <= base THEN
				faktor := base / v_plc_ticks_per_sec;
				MODE := FALSE;
			ELSE
				faktor := v_plc_ticks_per_sec / base;
				MODE := TRUE;
			END_IF;
		ELSE
			faktor := UDINT#1;
		END_IF;
		init := TRUE;
	END_IF;

	IF MODE THEN
		IF MODE THEN
		    T_PLC_MS := DINT_TO_UDINT(PLC_SYS_TICK_CNT) * faktor;
		ELSE
		    T_PLC_MS := DINT_TO_UDINT(PLC_SYS_TICK_CNT) / faktor;
		END_IF;
	ELSE
		T_PLC_MS := DINT_TO_UDINT(PLC_SYS_TICK_CNT) * faktor;
	END_IF;

	IF debug THEN
		T_PLC_MS := (DWORD_TO_UDINT(SHL(UDINT_TO_DWORD(T_PLC_MS),N) OR SHL(temp,N)) - UDINT#1) + Offset;
	END_IF;

END_FUNCTION_BLOCK

FUNCTION MODR : REAL
  VAR_INPUT
    IN : REAL;
    DIVI : REAL;
  END_VAR

  IF DIVI = 0.0 THEN
  	MODR := 0.0;
  ELSE
  	MODR := IN - DINT_TO_REAL(FLOOR2(IN / DIVI)) * DIVI;
  END_IF;
END_FUNCTION

FUNCTION FLOOR2 : DINT
  VAR_INPUT
    X : REAL;
  END_VAR

  FLOOR2 := REAL_TO_DINT(X);
  IF DINT_TO_REAL(FLOOR2) > X THEN
  	FLOOR2 := FLOOR2 - DINT#1;
  END_IF;
END_FUNCTION

FUNCTION _REAL_TO_DWORD: DWORD

  VAR_INPUT
    X :	REAL;
  END_VAR

  IF REAL_TO_DWORD(0.5) = DWORD#1 THEN
    _REAL_TO_DWORD := REAL_TO_DWORD(X);
  ELSIF X > 0.0 THEN
    _REAL_TO_DWORD := REAL_TO_DWORD(X+0.5);
  ELSIF X < 0.0 THEN
    _REAL_TO_DWORD := REAL_TO_DWORD(X-0.5);
  ELSE
    _REAL_TO_DWORD := DWORD#0;
  END_IF;
END_FUNCTION

FUNCTION _DWORD_TO_REAL:REAL
	VAR_INPUT
		IN :	DWORD;
	END_VAR

	_DWORD_TO_REAL := UDINT_TO_REAL(DWORD_TO_UDINT(IN));

END_FUNCTION

FUNCTION MULTIME_B:TIME
	VAR_INPUT
		T :	TIME;
		M :	REAL;
	END_VAR

	MULTIME_B := DWORD_TO_TIME(_REAL_TO_DWORD(_DWORD_TO_REAL(TIME_TO_DWORD(T))*M));
END_FUNCTION

FUNCTION_BLOCK GEN_SQR_Block

	VAR_INPUT
		PT :	TIME;
		AM :	REAL := REAL#1.0;
		OS :	REAL;
		DC :	REAL := REAL#0.5;
		DL :	REAL;
	END_VAR

	VAR_OUTPUT
		Q :	BOOL;
		Out :	REAL;
	END_VAR

	VAR
		TX :	TIME;
		last :	TIME;
		init :	BOOL;
		DLL: REAL;
		DCC: REAL;
		T_PLC_MS :	T_PLC_MS_block;
	END_VAR

	IF DC = 0.0 THEN
		Out := -AM * 0.5 + OS;
		Q := FALSE;
		RETURN;
	ELSIF DC = 1.0 THEN
		Out := AM * 0.5 + OS;
		Q := TRUE;
		RETURN;
	END_IF;

	T_PLC_MS();
	TX:= SUB_TIME(UDINT_TO_TIME(T_PLC_MS.T_PLC_MS) , last);
	DLL := MODR(DL,1.0);
	IF DLL < 0.0 THEN DLL := 1.0 - DLL; END_IF;
	DCC := MODR(DC,1.0);
	IF DCC < 0.0 THEN DCC := 1.0 - DCC; END_IF;

	IF NOT init THEN
		init := TRUE;
		last := TX;
		TX := t#0s;
	END_IF;

	IF TX >= PT THEN
		last := ADD_TIME( last , PT);
		TX := SUB_TIME(TX, PT);
	END_IF;

	IF MULTIME_B(PT, DL + DC) >= PT THEN
		IF TX >= MULTIME_B(PT, DL + DC - 1.0) THEN
			Out := -AM * 0.5 + OS;
			Q := FALSE;
		END_IF;
		IF TX >= MULTIME_B(PT, DL) THEN
			Out := AM * 0.5 + OS;
			Q := TRUE;
		END_IF;
	ELSE
		IF TX >= MULTIME_B(PT, DL) THEN
			Out := AM * 0.5 + OS;
			Q := TRUE;
		END_IF;
		IF TX >= MULTIME_B(PT, DL + DC) THEN
			Out := -AM * 0.5 + OS;
			Q := FALSE;
		END_IF;
	END_IF;

END_FUNCTION_BLOCK

PROGRAM program0
  VAR
	PT :	TIME;
	AM :	REAL := REAL#1.0;
	OS :	REAL;
	DC :	REAL := REAL#0.5;
	DL :	REAL;
	Q :	BOOL;
	Out :	REAL;
	func_block : GEN_SQR_Block;
  END_VAR
	func_block.PT  :=PT;
	func_block.AM  :=AM;
	func_block.OS  :=OS;
	func_block.DC  :=DC;
	func_block.DL  :=DL;
	func_block();
	Q := func_block.Q;
	Out := func_block.Out;
END_PROGRAM

(* ---- lb_claude_assisted_d74c0535eee0_0012.st ---- *)
TYPE
	oscat_parset_X              : ARRAY [1..4]    OF REAL;
	oscat_parset                : ARRAY [0..3]    OF oscat_parset_X := [0,0,0,0];
END_TYPE

FUNCTION TIME_TO_UDINT2:UDINT
	VAR_INPUT
		X :	TIME;
	END_VAR

	TIME_TO_UDINT2 := DINT_TO_UDINT(TIME_TO_DINT(X));
END_FUNCTION

FUNCTION _BYTE_TO_INT:INT
	VAR_INPUT
		IN :	BYTE;
	END_VAR

	_BYTE_TO_INT := USINT_TO_INT(BYTE_TO_USINT(IN));
END_FUNCTION

FUNCTION BIT_OF_DWORD : BOOL
  VAR_INPUT
    IN : DWORD;
    N : INT;
  END_VAR

  BIT_OF_DWORD := (SHR(in,N) AND 16#00000001) > 0;
  (* from OSCAT library; www.oscat.de  *)
END_FUNCTION

FUNCTION BIT_LOAD_B:BYTE
	VAR_INPUT
		IN :	BYTE;
		VAL :	BOOL;
		POS :	INT;
	END_VAR

	IF VAL THEN
		BIT_LOAD_B := in OR SHL(BYTE#1,pos);
	ELSE
		BIT_LOAD_B := in AND (NOT SHL(BYTE#1,pos));
	END_IF;
END_FUNCTION

FUNCTION_BLOCK T_PLC_MS_block
	VAR_OUTPUT
		T_PLC_MS :	UDINT;
	END_VAR

	VAR_EXTERNAL
		PLC_TICKS_PER_SEC :	INT;
		PLC_SYS_TICK_CNT :	DINT;
	END_VAR

	VAR
		debug :	BOOL;(*Debug-Mode ON / OFF*)
		N :	INT;(*Debug-Faktor*)
		Offset :	UDINT;(*Debug-Offset*)
		temp :	DWORD := DWORD#1;(*Debug-Offset*)
		mode :	BOOL;(*modus*)
		faktor :	UDINT;(*Systemtakt-Faktor*)
		init :	BOOL;
		v_plc_ticks_per_sec :	UDINT;
		base :	UDINT := UDINT#1000;
	END_VAR

	IF init = FALSE THEN
		v_plc_ticks_per_sec := INT_TO_UDINT(PLC_TICKS_PER_SEC);
		IF v_plc_ticks_per_sec = UDINT#1024 THEN
			faktor := UDINT#1;
			mode := FALSE;
		ELSIF v_plc_ticks_per_sec > UDINT#0 THEN
			IF v_plc_ticks_per_sec <= base THEN
				faktor := base / v_plc_ticks_per_sec;
				mode := FALSE;
			ELSE
				faktor := v_plc_ticks_per_sec / base;
				mode := TRUE;
			END_IF;
		ELSE
			faktor := UDINT#1;
		END_IF;
		init := TRUE;
	END_IF;

	IF mode THEN
		T_PLC_MS := DINT_TO_UDINT(PLC_SYS_TICK_CNT) / faktor;
	ELSE
		T_PLC_MS := DINT_TO_UDINT(PLC_SYS_TICK_CNT) * faktor;
	END_IF;

	IF debug THEN
		T_PLC_MS := (DWORD_TO_UDINT(SHL(UDINT_TO_DWORD(T_PLC_MS),N) OR SHL(temp,N)) - UDINT#1) + Offset;
	END_IF;
END_FUNCTION_BLOCK

FUNCTION_BLOCK PARSET_Block

	VAR_INPUT
		A0 :	BOOL;
		A1 :	BOOL;
		X01 :	REAL;
		X02 :	REAL;
		X03 :	REAL;
		X04 :	REAL;
		X11 :	REAL;
		X12 :	REAL;
		X13 :	REAL;
		X14 :	REAL;
		X21 :	REAL;
		X22 :	REAL;
		X23 :	REAL;
		X24 :	REAL;
		X31 :	REAL;
		X32 :	REAL;
		X33 :	REAL;
		X34 :	REAL;
		TC :	TIME;
	END_VAR

	VAR_OUTPUT
		P1 :	REAL;
		P2 :	REAL;
		P3 :	REAL;
		P4 :	REAL;
	END_VAR

	VAR
		X :	oscat_parset;
		S1 :	REAL;
		S2 :	REAL;
		S3 :	REAL;
		S4 :	REAL;
		tx :	UDINT;
		last :	UDINT;
		start :	BOOL;
		set :	BYTE;
		set2 :	INT;
		init :	BOOL;
		T_PLC_MS :	T_PLC_MS_Block;
	END_VAR

	(*@KEY@: WORKSHEET
	NAME: PARSET
	IEC_LANGUAGE: ST
	*)
	(* read system_time *)
	T_PLC_MS();
	tx:= T_PLC_MS.T_PLC_MS;

	(* init sequence *)
	IF NOT init THEN
		set:=BIT_LOAD_B(set,NOT A0,0); (* set.X0 := NOT A0; *)
		init := TRUE;
		X[0][1] := X01;
		X[0][2] := X02;
		X[0][3] := X03;
		X[0][4] := X04;
		X[1][1] := X11;
		X[1][2] := X12;
		X[1][3] := X13;
		X[1][4] := X14;
		X[2][1] := X21;
		X[2][2] := X22;
		X[2][3] := X23;
		X[2][4] := X24;
		X[3][1] := X31;
		X[3][2] := X32;
		X[3][3] := X33;
		X[3][4] := X34;
		P1 := X01;
		P2 := X02;
		P3 := X03;
		P4 := X04;
	END_IF;

	(* check for input change *)
	IF (A0 XOR BIT_OF_DWORD(BYTE_TO_DWORD(set),0)) OR (A1 XOR BIT_OF_DWORD(BYTE_TO_DWORD(set),1)) THEN  (* set.X0  ,  set.X1 *)
		(* a new set is selected *)
		set := BIT_LOAD_B(set,A0,0); (* set.X0 := A0; *)
		set := BIT_LOAD_B(set,A1,1); (* set.X1 := A1; *)

		IF tc > t#0s THEN
			start := TRUE;
			last := tx;
			(* save the step speed for the output changes in S *)
			set2 := _BYTE_TO_INT(set);
			S1 := (X[set2][1] - P1)/TIME_TO_REAL(tc);
			S2 := (X[set2][2] - P2)/TIME_TO_REAL(tc);
			S3 := (X[set2][3] - P3)/TIME_TO_REAL(tc);
			S4 := (X[set2][4] - P4)/TIME_TO_REAL(tc);
		END_IF;
	ELSIF start AND tx - last < TIME_TO_UDINT2(tc) THEN
		(* ramp the outputs to the new value *)
		set2 := _BYTE_TO_INT(set);
		P1 := X[set2][1] - S1*(TIME_TO_REAL(Tc) - UDINT_TO_REAL(tx + last));
		P2 := X[set2][2] - S2*(TIME_TO_REAL(Tc) - UDINT_TO_REAL(tx + last));
		P3 := X[set2][3] - S3*(TIME_TO_REAL(Tc) - UDINT_TO_REAL(tx + last));
		P4 := X[set2][4] - S4*(TIME_TO_REAL(Tc) - UDINT_TO_REAL(tx + last));
	ELSE
		(* make sure outputs match the correct set values *)
		set2 := _BYTE_TO_INT(set);
		IF start AND tx - last < TIME_TO_UDINT2(tc) THEN
		    start := TRUE;
		ELSE
		    start := FALSE;
		END_IF;
		P1 := X[set2][1];
		P2 := X[set2][2];
		P3 := X[set2][3];
		P4 := X[set2][4];
	END_IF;

END_FUNCTION_BLOCK

PROGRAM program0

	VAR
		A0 :	BOOL;
		A1 :	BOOL;
		X01 :	REAL;
		X02 :	REAL;
		X03 :	REAL;
		X04 :	REAL;
		X11 :	REAL;
		X12 :	REAL;
		X13 :	REAL;
		X14 :	REAL;
		X21 :	REAL;
		X22 :	REAL;
		X23 :	REAL;
		X24 :	REAL;
		X31 :	REAL;
		X32 :	REAL;
		X33 :	REAL;
		X34 :	REAL;
		TC :	TIME;

		P1 :	REAL;
		P2 :	REAL;
		P3 :	REAL;
		P4 :	REAL;
		func_block : PARSET_Block;
  	END_VAR
	func_block.A0 := A0;
	func_block.A1 := A1;
	func_block.X01 := X01;
	func_block.X02 := X02;
	func_block.X03 := X03;
	func_block.X04 := X04;
	func_block.X11 := X11;
	func_block.X12 := X12;
	func_block.X13 := X13;
	func_block.X14 := X14;
	func_block.X21 := X21;
	func_block.X22 := X22;
	func_block.X23 := X23;
	func_block.X24 := X24;
	func_block.X31 := X31;
	func_block.X32 := X32;
	func_block.X33 := X33;
	func_block.X34 := X34;
	func_block.TC := TC;
	func_block();
	P1 := func_block.P1;
	P2 := func_block.P2;
	P3 := func_block.P3;
	P4 := func_block.P4;

END_PROGRAM

CONFIGURATION Config0

	VAR_GLOBAL
		PLC_TICKS_PER_SEC :	INT;
		PLC_SYS_TICK_CNT :	DINT;
	END_VAR

  	RESOURCE Res0 ON PLC
    	TASK task0(INTERVAL := T#20ms,PRIORITY := 0);
    	PROGRAM instance0 WITH task0 : program0;
  	END_RESOURCE

END_CONFIGURATION

(* ---- lb_claude_assisted_d9c50a14bd9a_0117.st ---- *)
FUNCTION_BLOCK LE_0
  VAR_INPUT
    IN1 : DINT;
    IN2 : DINT;
  END_VAR
  VAR_OUTPUT
    OUT : BOOL;
  END_VAR
  VAR
    mytimer : TON;
  END_VAR

  OUT:=FALSE;
  IF IN1<=IN2 then
    OUT:=TRUE;
  END_IF;
  IF mytimer.Q = TRUE THEN
      mytimer(IN := TRUE, PT := T#9999h);
  ELSE
      mytimer(IN := TRUE, PT := t#8000ms);
  END_IF;

  IF mytimer.Q = TRUE then

      OUT:=TRUE;

  End_IF;
END_FUNCTION_BLOCK

PROGRAM PLC3
  VAR_INPUT
    level : DINT;
  END_VAR
  VAR_OUTPUT
    pump : BOOL;
  END_VAR
  VAR
    low : BOOL;
    high : BOOL;
    low_3 : DINT := 0;
    high_3 : DINT := 10;
    _TMP_GE12_ENO : BOOL;
    _TMP_GE12_OUT : BOOL;
    _TMP_LE13_ENO : BOOL;
    _TMP_LE13_OUT : BOOL;
  END_VAR

  _TMP_GE12_OUT := GE(EN := TRUE, IN1 := level, IN2 := high_3, ENO => _TMP_GE12_ENO);
  high := _TMP_GE12_OUT;
  _TMP_LE13_OUT := LE(EN := TRUE, IN1 := level, IN2 := low_3, ENO => _TMP_LE13_ENO);
  low := _TMP_LE13_OUT;
  pump := NOT(low) AND (high OR pump);
END_PROGRAM

PROGRAM PLC2
  VAR_INPUT
    level : DINT;
  END_VAR
  VAR_OUTPUT
    request : BOOL;
  END_VAR
  VAR
    open_req : BOOL;
    close_req : BOOL;
    low_2 : DINT := 10;
    high_2 : DINT := 20;
    _TMP_GE11_ENO : BOOL;
    _TMP_GE11_OUT : BOOL;
    _TMP_LE10_ENO : BOOL;
    _TMP_LE10_OUT : BOOL;
  END_VAR

  _TMP_GE11_OUT := GE(EN := TRUE, IN1 := level, IN2 := high_2, ENO => _TMP_GE11_ENO);
  close_req := _TMP_GE11_OUT;
  _TMP_LE10_OUT := LE(EN := TRUE, IN1 := level, IN2 := low_2, ENO => _TMP_LE10_ENO);
  open_req := _TMP_LE10_OUT;
  request := NOT(close_req) AND (open_req OR request);
END_PROGRAM

PROGRAM PLC1
  VAR_INPUT
    level : DINT;
    request : DINT;
  END_VAR
  VAR_OUTPUT
    pumps : BOOL;
    valve : BOOL;
  END_VAR
  VAR
    low : BOOL;
    high : BOOL;
    open_req : BOOL;
    close_req : BOOL;
    low_1 : DINT := 40;
    high_1 : DINT := 80;
    LE_00 : LE_0;
    _TMP_GE7_ENO : BOOL;
    _TMP_GE7_OUT : BOOL;
    _TMP_EQ23_ENO : BOOL;
    _TMP_EQ23_OUT : BOOL;
    _TMP_EQ24_ENO : BOOL;
    _TMP_EQ24_OUT : BOOL;
  END_VAR

  _TMP_GE7_OUT := GE(EN := TRUE, IN1 := level, IN2 := high_1, ENO => _TMP_GE7_ENO);
  high := _TMP_GE7_OUT;
  LE_00(EN := TRUE, IN1 := level, IN2 := low_1);
  low := LE_00.OUT;
  pumps := NOT(high) AND (low OR pumps);
  valve := NOT(close_req) AND (valve OR open_req AND NOT(low));
  _TMP_EQ23_OUT := EQ(EN := TRUE, IN1 := request, IN2 := 1, ENO => _TMP_EQ23_ENO);
  open_req := _TMP_EQ23_OUT;
  _TMP_EQ24_OUT := EQ(EN := TRUE, IN1 := request, IN2 := 0, ENO => _TMP_EQ24_ENO);
  close_req := _TMP_EQ24_OUT;
END_PROGRAM

CONFIGURATION Config0

  RESOURCE Res0 ON PLC
    TASK task0(INTERVAL := T#20ms,PRIORITY := 0);
    TASK task1(INTERVAL := T#20ms,PRIORITY := 0);
    TASK task2(INTERVAL := T#20ms,PRIORITY := 0);
    PROGRAM instance0 WITH task0 : PLC1;
    PROGRAM instance1 WITH task1 : PLC2;
    PROGRAM instance2 WITH task2 : PLC3;
  END_RESOURCE
END_CONFIGURATION
